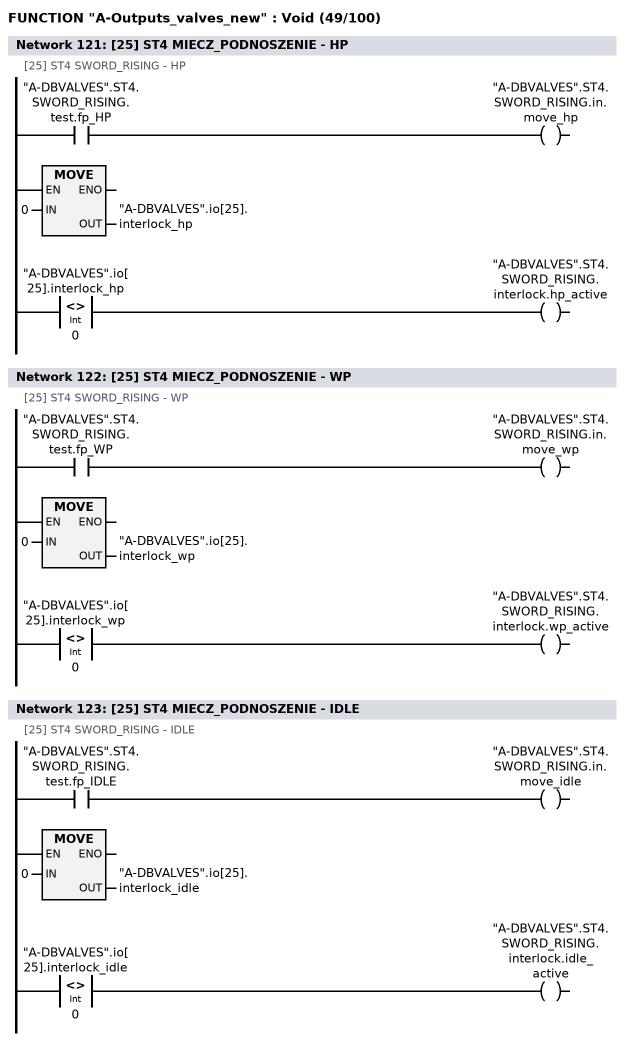
      O "A-DBVALVES".ST4.SWORD_RISING.test.fp_HP;
//    O     "A-Flags".STATION.IN_HP_STEP
      = "A-DBVALVES".ST4.SWORD_RISING.in.move_hp;

// Interlock hp
      L 0;
      T "A-DBVALVES".io[25].interlock_hp;

//{INTERLOCK_HP25}

      A(;
      L "A-DBVALVES".io[25].interlock_hp;
      L 0;
      <>I;
      );
      = "A-DBVALVES".ST4.SWORD_RISING.interlock.hp_active;
NETWORK
TITLE = [25] ST4 MIECZ_PODNOSZENIE - WP
//[25] ST4 SWORD_RISING - WP
      O "A-DBVALVES".ST4.SWORD_RISING.test.fp_WP;
      = "A-DBVALVES".ST4.SWORD_RISING.in.move_wp;

// Interlock wp
      L 0;
      T "A-DBVALVES".io[25].interlock_wp;

//{INTERLOCK_WP25}

      A(;
      L "A-DBVALVES".io[25].interlock_wp;
      L 0;
      <>I;
      );
      = "A-DBVALVES".ST4.SWORD_RISING.interlock.wp_active;
NETWORK
TITLE = [25] ST4 MIECZ_PODNOSZENIE - IDLE
//[25] ST4 SWORD_RISING - IDLE
      O "A-DBVALVES".ST4.SWORD_RISING.test.fp_IDLE;
      = "A-DBVALVES".ST4.SWORD_RISING.in.move_idle;

// Interlock idle
      L 0;
      T "A-DBVALVES".io[25].interlock_idle;

//{INTERLOCK_IDLE25}

      A(;
      L "A-DBVALVES".io[25].interlock_idle;
      L 0;
      <>I;
      );
      = "A-DBVALVES".ST4.SWORD_RISING.interlock.idle_active;
NETWORK
TITLE = [25] ST4 MIECZ_PODNOSZENIE
//[25] ST4 SWORD_RISING
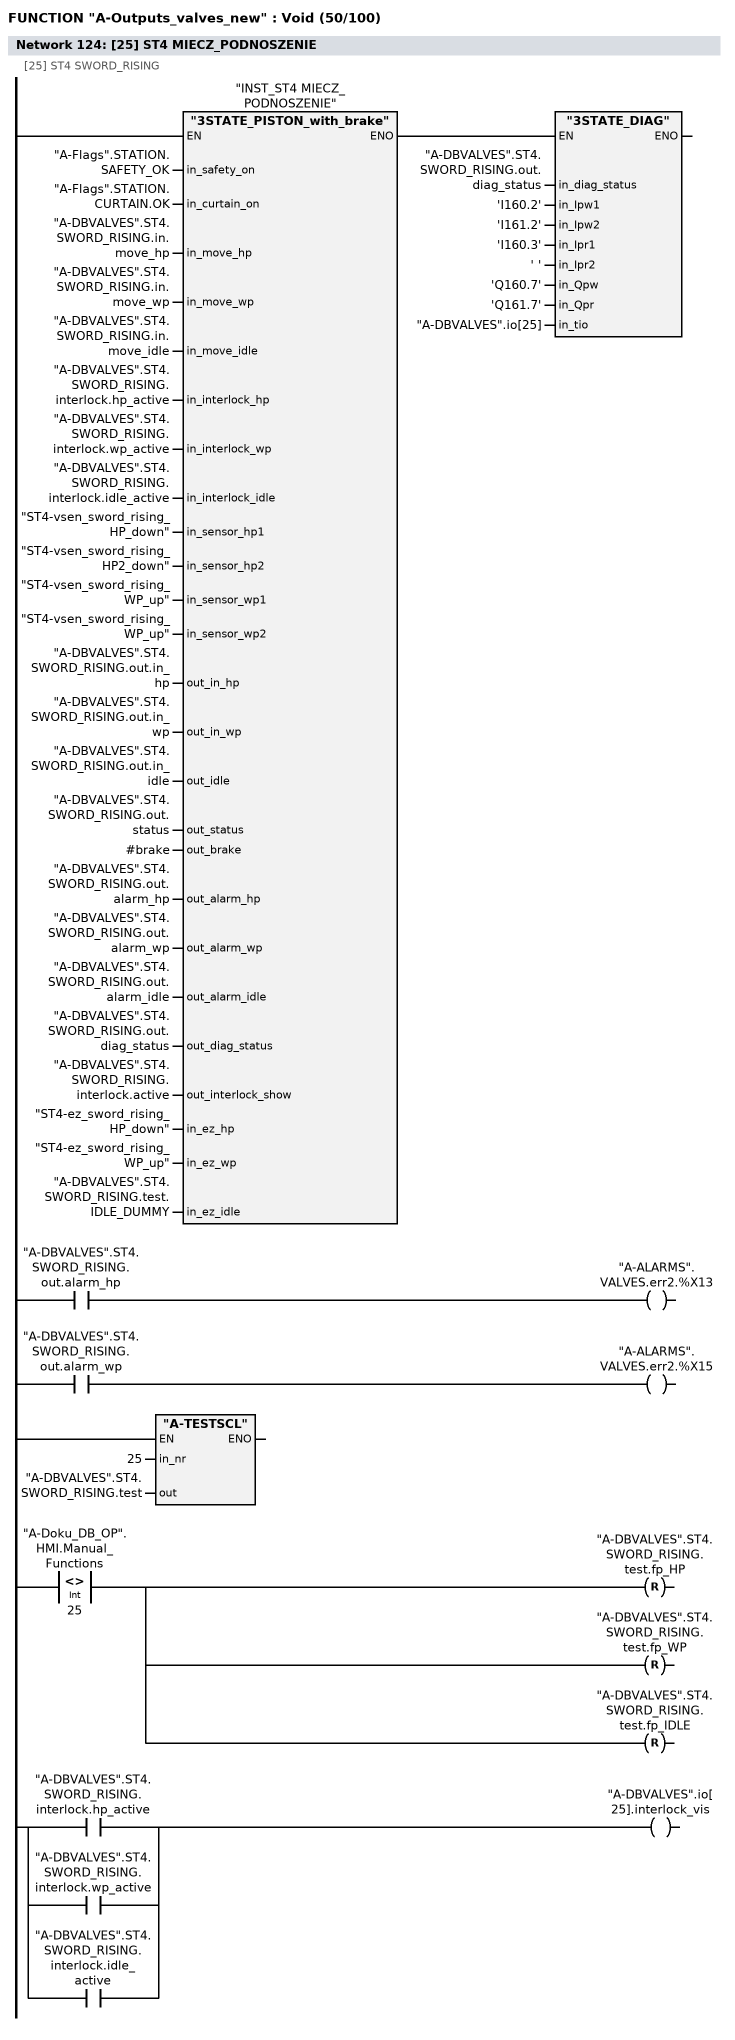
      CALL "3STATE_PISTON_with_brake", "INST_ST4 MIECZ_PODNOSZENIE"
      (  in_safety_on                := "A-Flags".STATION.SAFETY_OK ,
         in_curtain_on               := "A-Flags".STATION.CURTAIN.OK ,
         in_move_hp                  := "A-DBVALVES".ST4.SWORD_RISING.in.move_hp ,
         in_move_wp                  := "A-DBVALVES".ST4.SWORD_RISING.in.move_wp ,
         in_move_idle                := "A-DBVALVES".ST4.SWORD_RISING.in.move_idle ,
         in_interlock_hp             := "A-DBVALVES".ST4.SWORD_RISING.interlock.hp_active ,
         in_interlock_wp             := "A-DBVALVES".ST4.SWORD_RISING.interlock.wp_active ,
         in_interlock_idle           := "A-DBVALVES".ST4.SWORD_RISING.interlock.idle_active ,
         in_sensor_hp1               := "ST4-vsen_sword_rising_HP_down" ,
         in_sensor_hp2               := "ST4-vsen_sword_rising_HP2_down" ,
         in_sensor_wp1               := "ST4-vsen_sword_rising_WP_up" ,
         in_sensor_wp2               := "ST4-vsen_sword_rising_WP_up" ,
         out_in_hp                   := "A-DBVALVES".ST4.SWORD_RISING.out.in_hp ,
         out_in_wp                   := "A-DBVALVES".ST4.SWORD_RISING.out.in_wp ,
         out_idle                    := "A-DBVALVES".ST4.SWORD_RISING.out.in_idle ,
         out_status                  := "A-DBVALVES".ST4.SWORD_RISING.out.status ,
         out_brake                   := #brake ,
         out_alarm_hp                := "A-DBVALVES".ST4.SWORD_RISING.out.alarm_hp ,
         out_alarm_wp                := "A-DBVALVES".ST4.SWORD_RISING.out.alarm_wp ,
         out_alarm_idle              := "A-DBVALVES".ST4.SWORD_RISING.out.alarm_idle ,
         out_diag_status             := "A-DBVALVES".ST4.SWORD_RISING.out.diag_status ,
         out_interlock_show          := "A-DBVALVES".ST4.SWORD_RISING.interlock.active ,
         in_ez_hp                    := "ST4-ez_sword_rising_HP_down" ,
         in_ez_wp                    := "ST4-ez_sword_rising_WP_up" ,
         in_ez_idle                  := "A-DBVALVES".ST4.SWORD_RISING.test.IDLE_DUMMY
      );

      CALL "3STATE_DIAG"
      (  in_diag_status              := "A-DBVALVES".ST4.SWORD_RISING.out.diag_status ,
         in_Ipw1                     := 'I160.2' ,
         in_Ipw2                     := 'I161.2' ,
         in_Ipr1                     := 'I160.3' ,
         in_Ipr2                     := ' ' ,
         in_Qpw                      := 'Q160.7' ,
         in_Qpr                      := 'Q161.7' ,
         in_tio                      := "A-DBVALVES".io[25]
      );

      A "A-DBVALVES".ST4.SWORD_RISING.out.alarm_hp;
      = "A-ALARMS".VALVES.err2.%X13;

      A "A-DBVALVES".ST4.SWORD_RISING.out.alarm_wp;
      = "A-ALARMS".VALVES.err2.%X15;

      CALL "A-TESTSCL"
      (  in_nr                       := 25 ,
         out                         := "A-DBVALVES".ST4.SWORD_RISING.test
      );

      A(;
      L "A-Doku_DB_OP".HMI.Manual_Functions;
      L 25;
      <>I;
      );
      R "A-DBVALVES".ST4.SWORD_RISING.test.fp_HP;
      R "A-DBVALVES".ST4.SWORD_RISING.test.fp_WP;
      R "A-DBVALVES".ST4.SWORD_RISING.test.fp_IDLE;

      O "A-DBVALVES".ST4.SWORD_RISING.interlock.hp_active;
      O "A-DBVALVES".ST4.SWORD_RISING.interlock.wp_active;
      O "A-DBVALVES".ST4.SWORD_RISING.interlock.idle_active;
      = "A-DBVALVES".io[25].interlock_vis;
NETWORK
TITLE = -

NETWORK
TITLE = [26] ST4 ZDERZAK - HP
//[26] ST4 BUMPER - HP
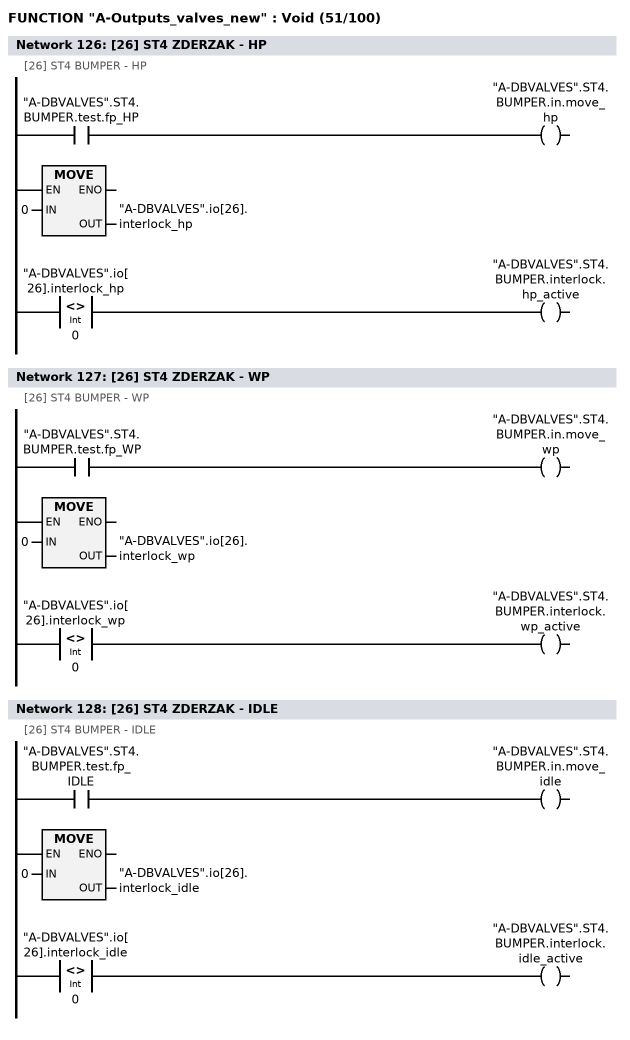
      O "A-DBVALVES".ST4.BUMPER.test.fp_HP;
//    O     "A-Flags".STATION.IN_HP_STEP
      = "A-DBVALVES".ST4.BUMPER.in.move_hp;

// Interlock hp
      L 0;
      T "A-DBVALVES".io[26].interlock_hp;

//{INTERLOCK_HP26}

      A(;
      L "A-DBVALVES".io[26].interlock_hp;
      L 0;
      <>I;
      );
      = "A-DBVALVES".ST4.BUMPER.interlock.hp_active;
NETWORK
TITLE = [26] ST4 ZDERZAK - WP
//[26] ST4 BUMPER - WP
      O "A-DBVALVES".ST4.BUMPER.test.fp_WP;
      = "A-DBVALVES".ST4.BUMPER.in.move_wp;

// Interlock wp
      L 0;
      T "A-DBVALVES".io[26].interlock_wp;

//{INTERLOCK_WP26}

      A(;
      L "A-DBVALVES".io[26].interlock_wp;
      L 0;
      <>I;
      );
      = "A-DBVALVES".ST4.BUMPER.interlock.wp_active;
NETWORK
TITLE = [26] ST4 ZDERZAK - IDLE
//[26] ST4 BUMPER - IDLE
      O "A-DBVALVES".ST4.BUMPER.test.fp_IDLE;
      = "A-DBVALVES".ST4.BUMPER.in.move_idle;

// Interlock idle
      L 0;
      T "A-DBVALVES".io[26].interlock_idle;

//{INTERLOCK_IDLE26}

      A(;
      L "A-DBVALVES".io[26].interlock_idle;
      L 0;
      <>I;
      );
      = "A-DBVALVES".ST4.BUMPER.interlock.idle_active;
NETWORK
TITLE = [26] ST4 ZDERZAK
//[26] ST4 BUMPER
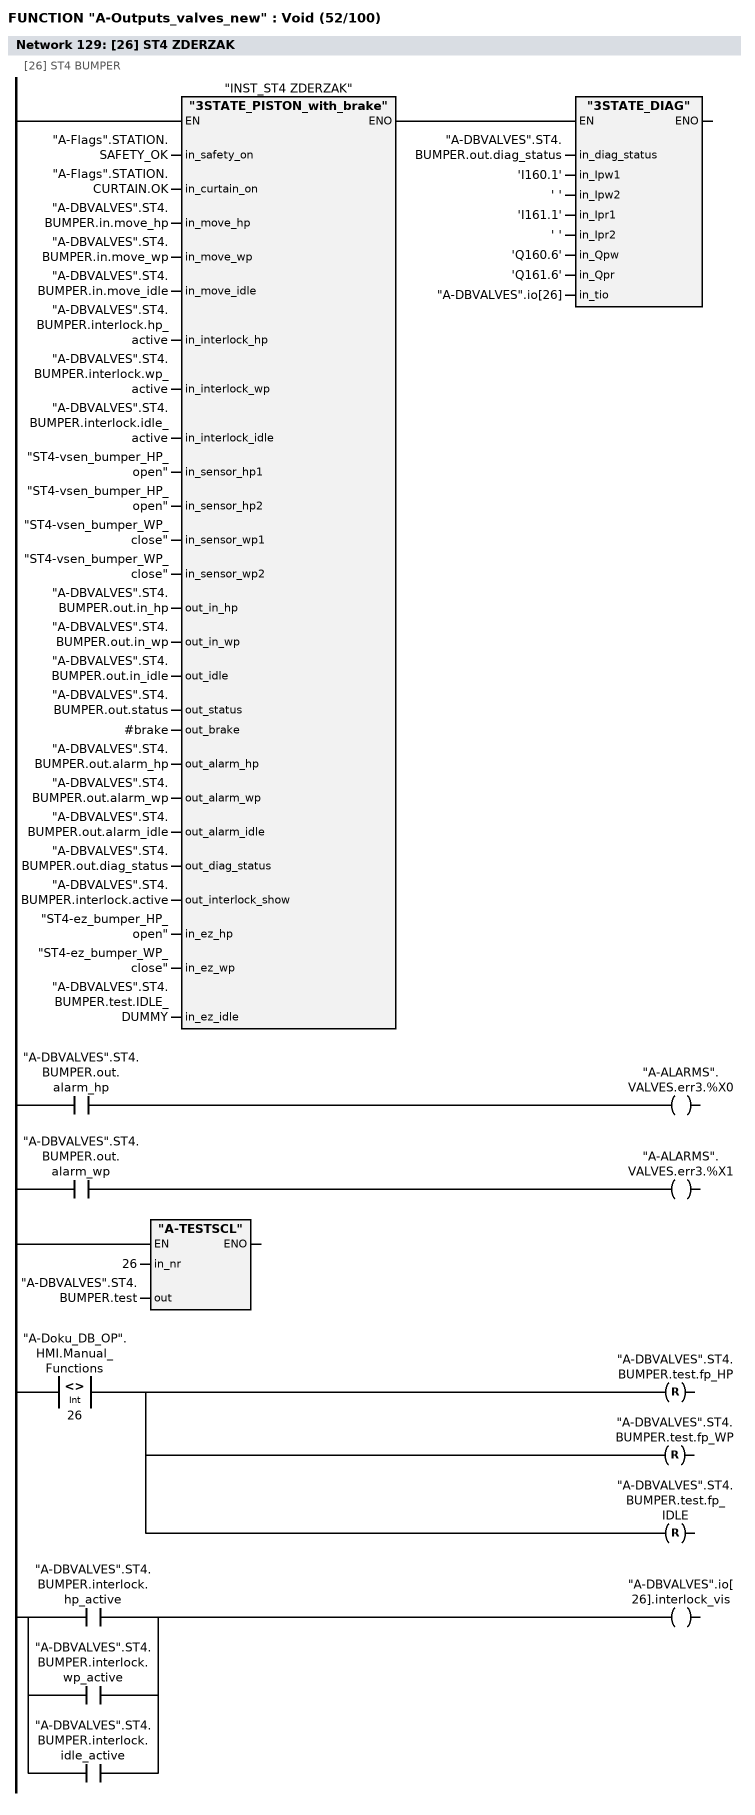
      CALL "3STATE_PISTON_with_brake", "INST_ST4 ZDERZAK"
      (  in_safety_on                := "A-Flags".STATION.SAFETY_OK ,
         in_curtain_on               := "A-Flags".STATION.CURTAIN.OK ,
         in_move_hp                  := "A-DBVALVES".ST4.BUMPER.in.move_hp ,
         in_move_wp                  := "A-DBVALVES".ST4.BUMPER.in.move_wp ,
         in_move_idle                := "A-DBVALVES".ST4.BUMPER.in.move_idle ,
         in_interlock_hp             := "A-DBVALVES".ST4.BUMPER.interlock.hp_active ,
         in_interlock_wp             := "A-DBVALVES".ST4.BUMPER.interlock.wp_active ,
         in_interlock_idle           := "A-DBVALVES".ST4.BUMPER.interlock.idle_active ,
         in_sensor_hp1               := "ST4-vsen_bumper_HP_open" ,
         in_sensor_hp2               := "ST4-vsen_bumper_HP_open" ,
         in_sensor_wp1               := "ST4-vsen_bumper_WP_close" ,
         in_sensor_wp2               := "ST4-vsen_bumper_WP_close" ,
         out_in_hp                   := "A-DBVALVES".ST4.BUMPER.out.in_hp ,
         out_in_wp                   := "A-DBVALVES".ST4.BUMPER.out.in_wp ,
         out_idle                    := "A-DBVALVES".ST4.BUMPER.out.in_idle ,
         out_status                  := "A-DBVALVES".ST4.BUMPER.out.status ,
         out_brake                   := #brake ,
         out_alarm_hp                := "A-DBVALVES".ST4.BUMPER.out.alarm_hp ,
         out_alarm_wp                := "A-DBVALVES".ST4.BUMPER.out.alarm_wp ,
         out_alarm_idle              := "A-DBVALVES".ST4.BUMPER.out.alarm_idle ,
         out_diag_status             := "A-DBVALVES".ST4.BUMPER.out.diag_status ,
         out_interlock_show          := "A-DBVALVES".ST4.BUMPER.interlock.active ,
         in_ez_hp                    := "ST4-ez_bumper_HP_open" ,
         in_ez_wp                    := "ST4-ez_bumper_WP_close" ,
         in_ez_idle                  := "A-DBVALVES".ST4.BUMPER.test.IDLE_DUMMY
      );

      CALL "3STATE_DIAG"
      (  in_diag_status              := "A-DBVALVES".ST4.BUMPER.out.diag_status ,
         in_Ipw1                     := 'I160.1' ,
         in_Ipw2                     := ' ' ,
         in_Ipr1                     := 'I161.1' ,
         in_Ipr2                     := ' ' ,
         in_Qpw                      := 'Q160.6' ,
         in_Qpr                      := 'Q161.6' ,
         in_tio                      := "A-DBVALVES".io[26]
      );

      A "A-DBVALVES".ST4.BUMPER.out.alarm_hp;
      = "A-ALARMS".VALVES.err3.%X0;

      A "A-DBVALVES".ST4.BUMPER.out.alarm_wp;
      = "A-ALARMS".VALVES.err3.%X1;

      CALL "A-TESTSCL"
      (  in_nr                       := 26 ,
         out                         := "A-DBVALVES".ST4.BUMPER.test
      );

      A(;
      L "A-Doku_DB_OP".HMI.Manual_Functions;
      L 26;
      <>I;
      );
      R "A-DBVALVES".ST4.BUMPER.test.fp_HP;
      R "A-DBVALVES".ST4.BUMPER.test.fp_WP;
      R "A-DBVALVES".ST4.BUMPER.test.fp_IDLE;

      O "A-DBVALVES".ST4.BUMPER.interlock.hp_active;
      O "A-DBVALVES".ST4.BUMPER.interlock.wp_active;
      O "A-DBVALVES".ST4.BUMPER.interlock.idle_active;
      = "A-DBVALVES".io[26].interlock_vis;
NETWORK
TITLE = -

NETWORK
TITLE = [27] ST4 MIECZ - HP
//[27] ST4 SWORD - HP
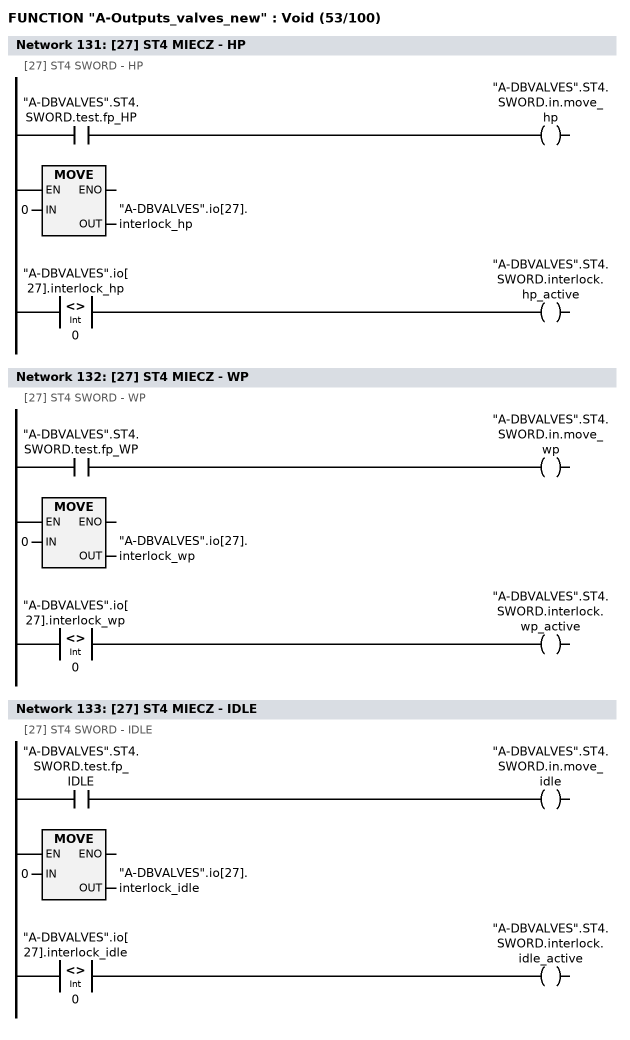
      O "A-DBVALVES".ST4.SWORD.test.fp_HP;
//    O     "A-Flags".STATION.IN_HP_STEP
      = "A-DBVALVES".ST4.SWORD.in.move_hp;

// Interlock hp
      L 0;
      T "A-DBVALVES".io[27].interlock_hp;

//{INTERLOCK_HP27}

      A(;
      L "A-DBVALVES".io[27].interlock_hp;
      L 0;
      <>I;
      );
      = "A-DBVALVES".ST4.SWORD.interlock.hp_active;
NETWORK
TITLE = [27] ST4 MIECZ - WP
//[27] ST4 SWORD - WP
      O "A-DBVALVES".ST4.SWORD.test.fp_WP;
      = "A-DBVALVES".ST4.SWORD.in.move_wp;

// Interlock wp
      L 0;
      T "A-DBVALVES".io[27].interlock_wp;

//{INTERLOCK_WP27}

      A(;
      L "A-DBVALVES".io[27].interlock_wp;
      L 0;
      <>I;
      );
      = "A-DBVALVES".ST4.SWORD.interlock.wp_active;
NETWORK
TITLE = [27] ST4 MIECZ - IDLE
//[27] ST4 SWORD - IDLE
      O "A-DBVALVES".ST4.SWORD.test.fp_IDLE;
      = "A-DBVALVES".ST4.SWORD.in.move_idle;

// Interlock idle
      L 0;
      T "A-DBVALVES".io[27].interlock_idle;

//{INTERLOCK_IDLE27}

      A(;
      L "A-DBVALVES".io[27].interlock_idle;
      L 0;
      <>I;
      );
      = "A-DBVALVES".ST4.SWORD.interlock.idle_active;
NETWORK
TITLE = [27] ST4 MIECZ
//[27] ST4 SWORD
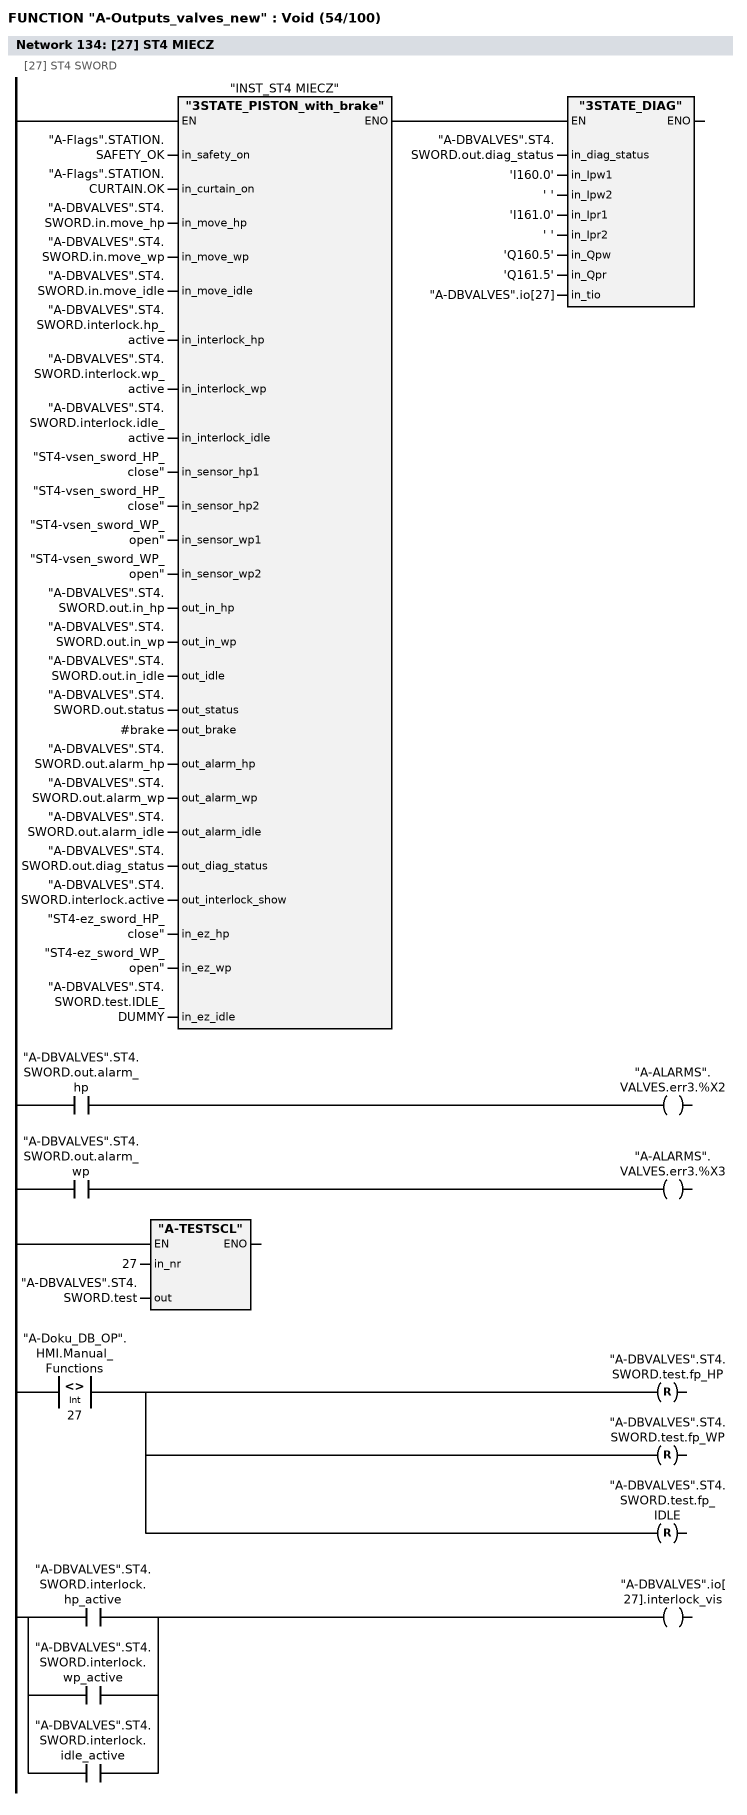
      CALL "3STATE_PISTON_with_brake", "INST_ST4 MIECZ"
      (  in_safety_on                := "A-Flags".STATION.SAFETY_OK ,
         in_curtain_on               := "A-Flags".STATION.CURTAIN.OK ,
         in_move_hp                  := "A-DBVALVES".ST4.SWORD.in.move_hp ,
         in_move_wp                  := "A-DBVALVES".ST4.SWORD.in.move_wp ,
         in_move_idle                := "A-DBVALVES".ST4.SWORD.in.move_idle ,
         in_interlock_hp             := "A-DBVALVES".ST4.SWORD.interlock.hp_active ,
         in_interlock_wp             := "A-DBVALVES".ST4.SWORD.interlock.wp_active ,
         in_interlock_idle           := "A-DBVALVES".ST4.SWORD.interlock.idle_active ,
         in_sensor_hp1               := "ST4-vsen_sword_HP_close" ,
         in_sensor_hp2               := "ST4-vsen_sword_HP_close" ,
         in_sensor_wp1               := "ST4-vsen_sword_WP_open" ,
         in_sensor_wp2               := "ST4-vsen_sword_WP_open" ,
         out_in_hp                   := "A-DBVALVES".ST4.SWORD.out.in_hp ,
         out_in_wp                   := "A-DBVALVES".ST4.SWORD.out.in_wp ,
         out_idle                    := "A-DBVALVES".ST4.SWORD.out.in_idle ,
         out_status                  := "A-DBVALVES".ST4.SWORD.out.status ,
         out_brake                   := #brake ,
         out_alarm_hp                := "A-DBVALVES".ST4.SWORD.out.alarm_hp ,
         out_alarm_wp                := "A-DBVALVES".ST4.SWORD.out.alarm_wp ,
         out_alarm_idle              := "A-DBVALVES".ST4.SWORD.out.alarm_idle ,
         out_diag_status             := "A-DBVALVES".ST4.SWORD.out.diag_status ,
         out_interlock_show          := "A-DBVALVES".ST4.SWORD.interlock.active ,
         in_ez_hp                    := "ST4-ez_sword_HP_close" ,
         in_ez_wp                    := "ST4-ez_sword_WP_open" ,
         in_ez_idle                  := "A-DBVALVES".ST4.SWORD.test.IDLE_DUMMY
      );

      CALL "3STATE_DIAG"
      (  in_diag_status              := "A-DBVALVES".ST4.SWORD.out.diag_status ,
         in_Ipw1                     := 'I160.0' ,
         in_Ipw2                     := ' ' ,
         in_Ipr1                     := 'I161.0' ,
         in_Ipr2                     := ' ' ,
         in_Qpw                      := 'Q160.5' ,
         in_Qpr                      := 'Q161.5' ,
         in_tio                      := "A-DBVALVES".io[27]
      );

      A "A-DBVALVES".ST4.SWORD.out.alarm_hp;
      = "A-ALARMS".VALVES.err3.%X2;

      A "A-DBVALVES".ST4.SWORD.out.alarm_wp;
      = "A-ALARMS".VALVES.err3.%X3;

      CALL "A-TESTSCL"
      (  in_nr                       := 27 ,
         out                         := "A-DBVALVES".ST4.SWORD.test
      );

      A(;
      L "A-Doku_DB_OP".HMI.Manual_Functions;
      L 27;
      <>I;
      );
      R "A-DBVALVES".ST4.SWORD.test.fp_HP;
      R "A-DBVALVES".ST4.SWORD.test.fp_WP;
      R "A-DBVALVES".ST4.SWORD.test.fp_IDLE;

      O "A-DBVALVES".ST4.SWORD.interlock.hp_active;
      O "A-DBVALVES".ST4.SWORD.interlock.wp_active;
      O "A-DBVALVES".ST4.SWORD.interlock.idle_active;
      = "A-DBVALVES".io[27].interlock_vis;
NETWORK
TITLE = -

NETWORK
TITLE = [28] ST5 STACJA_DOJAZD - HP
//[28] ST5 STATION_MOVEMENT - HP
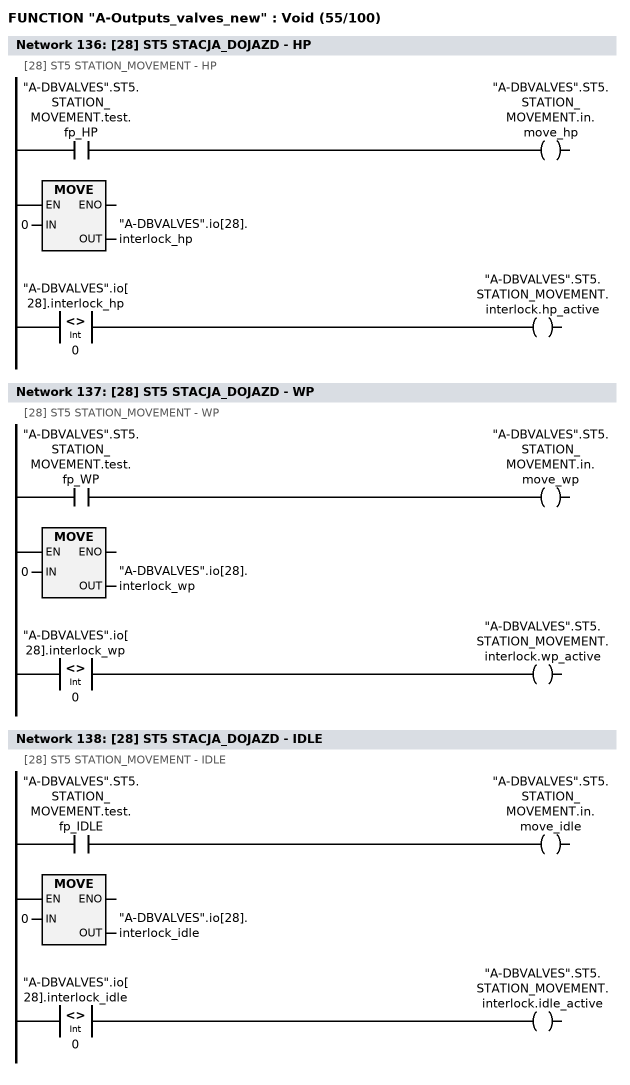
      O "A-DBVALVES".ST5.STATION_MOVEMENT.test.fp_HP;
//    O     "A-Flags".STATION.IN_HP_STEP
      = "A-DBVALVES".ST5.STATION_MOVEMENT.in.move_hp;

// Interlock hp
      L 0;
      T "A-DBVALVES".io[28].interlock_hp;

//{INTERLOCK_HP28}

      A(;
      L "A-DBVALVES".io[28].interlock_hp;
      L 0;
      <>I;
      );
      = "A-DBVALVES".ST5.STATION_MOVEMENT.interlock.hp_active;
NETWORK
TITLE = [28] ST5 STACJA_DOJAZD - WP
//[28] ST5 STATION_MOVEMENT - WP
      O "A-DBVALVES".ST5.STATION_MOVEMENT.test.fp_WP;
      = "A-DBVALVES".ST5.STATION_MOVEMENT.in.move_wp;

// Interlock wp
      L 0;
      T "A-DBVALVES".io[28].interlock_wp;

//{INTERLOCK_WP28}

      A(;
      L "A-DBVALVES".io[28].interlock_wp;
      L 0;
      <>I;
      );
      = "A-DBVALVES".ST5.STATION_MOVEMENT.interlock.wp_active;
NETWORK
TITLE = [28] ST5 STACJA_DOJAZD - IDLE
//[28] ST5 STATION_MOVEMENT - IDLE
      O "A-DBVALVES".ST5.STATION_MOVEMENT.test.fp_IDLE;
      = "A-DBVALVES".ST5.STATION_MOVEMENT.in.move_idle;

// Interlock idle
      L 0;
      T "A-DBVALVES".io[28].interlock_idle;

//{INTERLOCK_IDLE28}

      A(;
      L "A-DBVALVES".io[28].interlock_idle;
      L 0;
      <>I;
      );
      = "A-DBVALVES".ST5.STATION_MOVEMENT.interlock.idle_active;
NETWORK
TITLE = [28] ST5 STACJA_DOJAZD
//[28] ST5 STATION_MOVEMENT
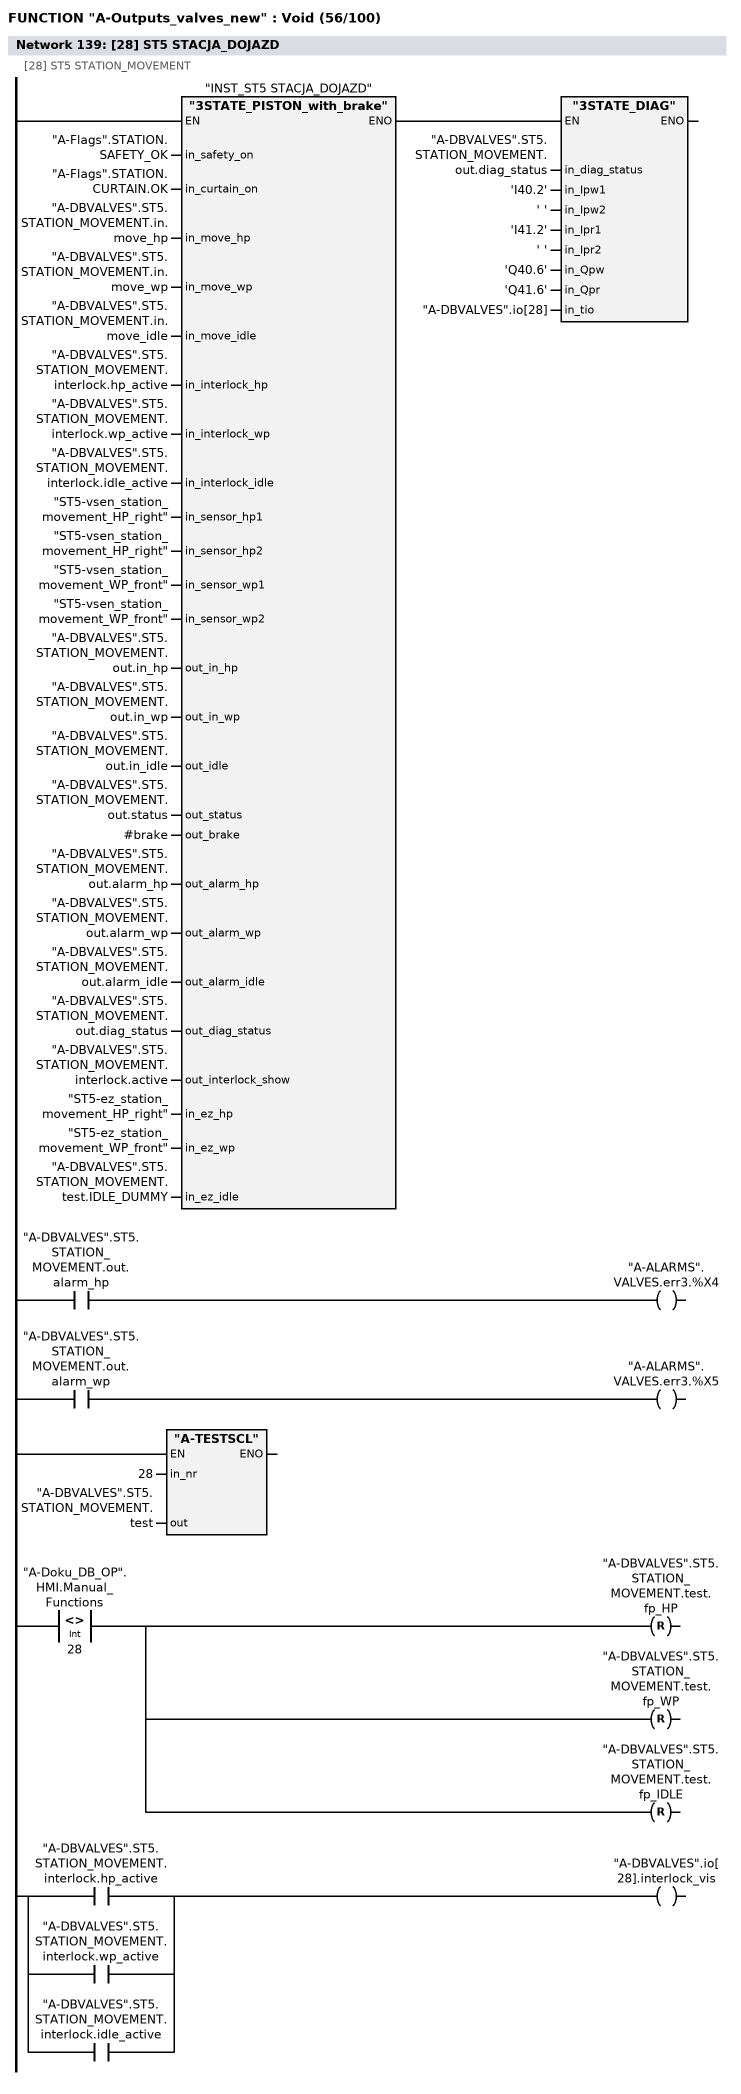
      CALL "3STATE_PISTON_with_brake", "INST_ST5 STACJA_DOJAZD"
      (  in_safety_on                := "A-Flags".STATION.SAFETY_OK ,
         in_curtain_on               := "A-Flags".STATION.CURTAIN.OK ,
         in_move_hp                  := "A-DBVALVES".ST5.STATION_MOVEMENT.in.move_hp ,
         in_move_wp                  := "A-DBVALVES".ST5.STATION_MOVEMENT.in.move_wp ,
         in_move_idle                := "A-DBVALVES".ST5.STATION_MOVEMENT.in.move_idle ,
         in_interlock_hp             := "A-DBVALVES".ST5.STATION_MOVEMENT.interlock.hp_active ,
         in_interlock_wp             := "A-DBVALVES".ST5.STATION_MOVEMENT.interlock.wp_active ,
         in_interlock_idle           := "A-DBVALVES".ST5.STATION_MOVEMENT.interlock.idle_active ,
         in_sensor_hp1               := "ST5-vsen_station_movement_HP_right" ,
         in_sensor_hp2               := "ST5-vsen_station_movement_HP_right" ,
         in_sensor_wp1               := "ST5-vsen_station_movement_WP_front" ,
         in_sensor_wp2               := "ST5-vsen_station_movement_WP_front" ,
         out_in_hp                   := "A-DBVALVES".ST5.STATION_MOVEMENT.out.in_hp ,
         out_in_wp                   := "A-DBVALVES".ST5.STATION_MOVEMENT.out.in_wp ,
         out_idle                    := "A-DBVALVES".ST5.STATION_MOVEMENT.out.in_idle ,
         out_status                  := "A-DBVALVES".ST5.STATION_MOVEMENT.out.status ,
         out_brake                   := #brake ,
         out_alarm_hp                := "A-DBVALVES".ST5.STATION_MOVEMENT.out.alarm_hp ,
         out_alarm_wp                := "A-DBVALVES".ST5.STATION_MOVEMENT.out.alarm_wp ,
         out_alarm_idle              := "A-DBVALVES".ST5.STATION_MOVEMENT.out.alarm_idle ,
         out_diag_status             := "A-DBVALVES".ST5.STATION_MOVEMENT.out.diag_status ,
         out_interlock_show          := "A-DBVALVES".ST5.STATION_MOVEMENT.interlock.active ,
         in_ez_hp                    := "ST5-ez_station_movement_HP_right" ,
         in_ez_wp                    := "ST5-ez_station_movement_WP_front" ,
         in_ez_idle                  := "A-DBVALVES".ST5.STATION_MOVEMENT.test.IDLE_DUMMY
      );

      CALL "3STATE_DIAG"
      (  in_diag_status              := "A-DBVALVES".ST5.STATION_MOVEMENT.out.diag_status ,
         in_Ipw1                     := 'I40.2' ,
         in_Ipw2                     := ' ' ,
         in_Ipr1                     := 'I41.2' ,
         in_Ipr2                     := ' ' ,
         in_Qpw                      := 'Q40.6' ,
         in_Qpr                      := 'Q41.6' ,
         in_tio                      := "A-DBVALVES".io[28]
      );

      A "A-DBVALVES".ST5.STATION_MOVEMENT.out.alarm_hp;
      = "A-ALARMS".VALVES.err3.%X4;

      A "A-DBVALVES".ST5.STATION_MOVEMENT.out.alarm_wp;
      = "A-ALARMS".VALVES.err3.%X5;

      CALL "A-TESTSCL"
      (  in_nr                       := 28 ,
         out                         := "A-DBVALVES".ST5.STATION_MOVEMENT.test
      );

      A(;
      L "A-Doku_DB_OP".HMI.Manual_Functions;
      L 28;
      <>I;
      );
      R "A-DBVALVES".ST5.STATION_MOVEMENT.test.fp_HP;
      R "A-DBVALVES".ST5.STATION_MOVEMENT.test.fp_WP;
      R "A-DBVALVES".ST5.STATION_MOVEMENT.test.fp_IDLE;

      O "A-DBVALVES".ST5.STATION_MOVEMENT.interlock.hp_active;
      O "A-DBVALVES".ST5.STATION_MOVEMENT.interlock.wp_active;
      O "A-DBVALVES".ST5.STATION_MOVEMENT.interlock.idle_active;
      = "A-DBVALVES".io[28].interlock_vis;
NETWORK
TITLE = -

NETWORK
TITLE = [29] ST5 STACJA_MALY_SKOK - HP
//[29] ST5 STATION_SMALL_STEP - HP
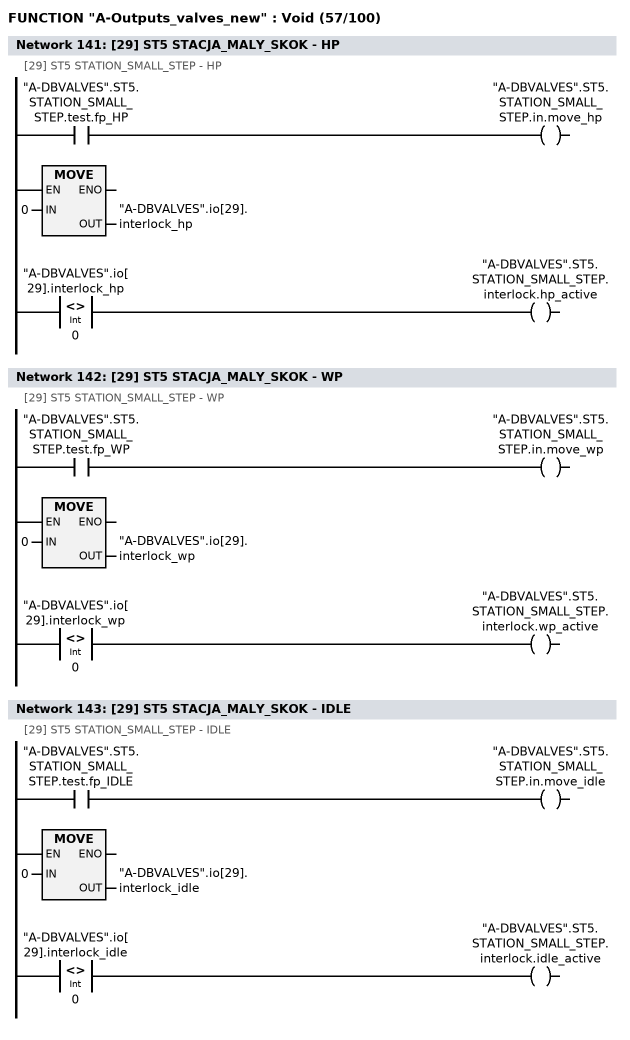
      O "A-DBVALVES".ST5.STATION_SMALL_STEP.test.fp_HP;
//    O     "A-Flags".STATION.IN_HP_STEP
      = "A-DBVALVES".ST5.STATION_SMALL_STEP.in.move_hp;

// Interlock hp
      L 0;
      T "A-DBVALVES".io[29].interlock_hp;

//{INTERLOCK_HP29}

      A(;
      L "A-DBVALVES".io[29].interlock_hp;
      L 0;
      <>I;
      );
      = "A-DBVALVES".ST5.STATION_SMALL_STEP.interlock.hp_active;
NETWORK
TITLE = [29] ST5 STACJA_MALY_SKOK - WP
//[29] ST5 STATION_SMALL_STEP - WP
      O "A-DBVALVES".ST5.STATION_SMALL_STEP.test.fp_WP;
      = "A-DBVALVES".ST5.STATION_SMALL_STEP.in.move_wp;

// Interlock wp
      L 0;
      T "A-DBVALVES".io[29].interlock_wp;

//{INTERLOCK_WP29}

      A(;
      L "A-DBVALVES".io[29].interlock_wp;
      L 0;
      <>I;
      );
      = "A-DBVALVES".ST5.STATION_SMALL_STEP.interlock.wp_active;
NETWORK
TITLE = [29] ST5 STACJA_MALY_SKOK - IDLE
//[29] ST5 STATION_SMALL_STEP - IDLE
      O "A-DBVALVES".ST5.STATION_SMALL_STEP.test.fp_IDLE;
      = "A-DBVALVES".ST5.STATION_SMALL_STEP.in.move_idle;

// Interlock idle
      L 0;
      T "A-DBVALVES".io[29].interlock_idle;

//{INTERLOCK_IDLE29}

      A(;
      L "A-DBVALVES".io[29].interlock_idle;
      L 0;
      <>I;
      );
      = "A-DBVALVES".ST5.STATION_SMALL_STEP.interlock.idle_active;
NETWORK
TITLE = [29] ST5 STACJA_MALY_SKOK
//[29] ST5 STATION_SMALL_STEP
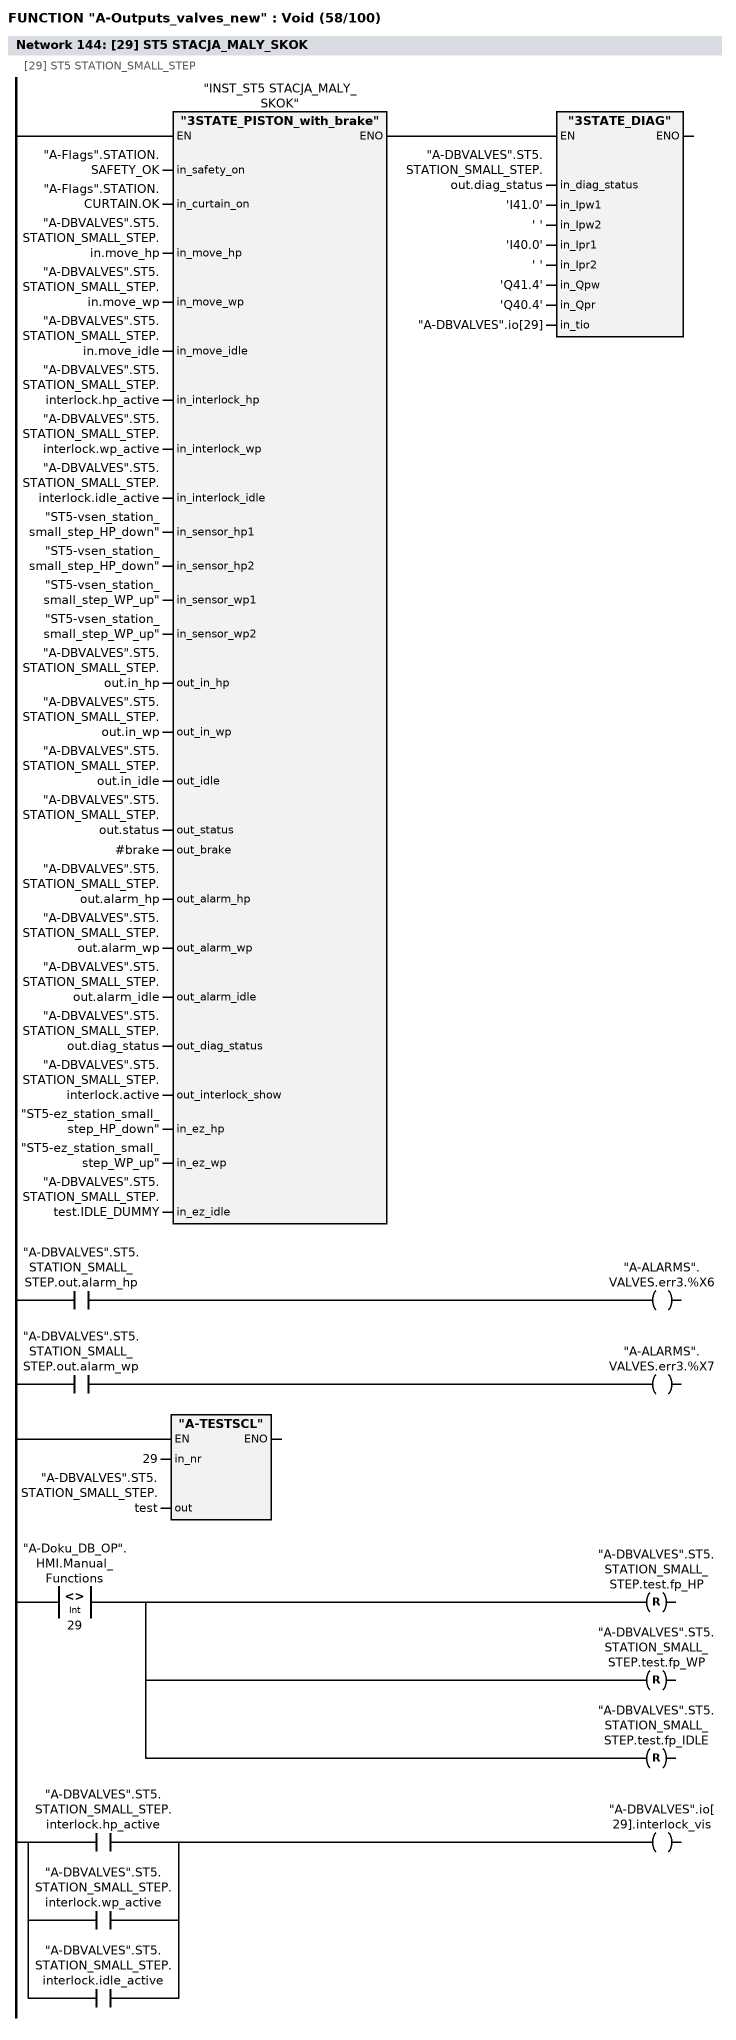
      CALL "3STATE_PISTON_with_brake", "INST_ST5 STACJA_MALY_SKOK"
      (  in_safety_on                := "A-Flags".STATION.SAFETY_OK ,
         in_curtain_on               := "A-Flags".STATION.CURTAIN.OK ,
         in_move_hp                  := "A-DBVALVES".ST5.STATION_SMALL_STEP.in.move_hp ,
         in_move_wp                  := "A-DBVALVES".ST5.STATION_SMALL_STEP.in.move_wp ,
         in_move_idle                := "A-DBVALVES".ST5.STATION_SMALL_STEP.in.move_idle ,
         in_interlock_hp             := "A-DBVALVES".ST5.STATION_SMALL_STEP.interlock.hp_active ,
         in_interlock_wp             := "A-DBVALVES".ST5.STATION_SMALL_STEP.interlock.wp_active ,
         in_interlock_idle           := "A-DBVALVES".ST5.STATION_SMALL_STEP.interlock.idle_active ,
         in_sensor_hp1               := "ST5-vsen_station_small_step_HP_down" ,
         in_sensor_hp2               := "ST5-vsen_station_small_step_HP_down" ,
         in_sensor_wp1               := "ST5-vsen_station_small_step_WP_up" ,
         in_sensor_wp2               := "ST5-vsen_station_small_step_WP_up" ,
         out_in_hp                   := "A-DBVALVES".ST5.STATION_SMALL_STEP.out.in_hp ,
         out_in_wp                   := "A-DBVALVES".ST5.STATION_SMALL_STEP.out.in_wp ,
         out_idle                    := "A-DBVALVES".ST5.STATION_SMALL_STEP.out.in_idle ,
         out_status                  := "A-DBVALVES".ST5.STATION_SMALL_STEP.out.status ,
         out_brake                   := #brake ,
         out_alarm_hp                := "A-DBVALVES".ST5.STATION_SMALL_STEP.out.alarm_hp ,
         out_alarm_wp                := "A-DBVALVES".ST5.STATION_SMALL_STEP.out.alarm_wp ,
         out_alarm_idle              := "A-DBVALVES".ST5.STATION_SMALL_STEP.out.alarm_idle ,
         out_diag_status             := "A-DBVALVES".ST5.STATION_SMALL_STEP.out.diag_status ,
         out_interlock_show          := "A-DBVALVES".ST5.STATION_SMALL_STEP.interlock.active ,
         in_ez_hp                    := "ST5-ez_station_small_step_HP_down" ,
         in_ez_wp                    := "ST5-ez_station_small_step_WP_up" ,
         in_ez_idle                  := "A-DBVALVES".ST5.STATION_SMALL_STEP.test.IDLE_DUMMY
      );

      CALL "3STATE_DIAG"
      (  in_diag_status              := "A-DBVALVES".ST5.STATION_SMALL_STEP.out.diag_status ,
         in_Ipw1                     := 'I41.0' ,
         in_Ipw2                     := ' ' ,
         in_Ipr1                     := 'I40.0' ,
         in_Ipr2                     := ' ' ,
         in_Qpw                      := 'Q41.4' ,
         in_Qpr                      := 'Q40.4' ,
         in_tio                      := "A-DBVALVES".io[29]
      );

      A "A-DBVALVES".ST5.STATION_SMALL_STEP.out.alarm_hp;
      = "A-ALARMS".VALVES.err3.%X6;

      A "A-DBVALVES".ST5.STATION_SMALL_STEP.out.alarm_wp;
      = "A-ALARMS".VALVES.err3.%X7;

      CALL "A-TESTSCL"
      (  in_nr                       := 29 ,
         out                         := "A-DBVALVES".ST5.STATION_SMALL_STEP.test
      );

      A(;
      L "A-Doku_DB_OP".HMI.Manual_Functions;
      L 29;
      <>I;
      );
      R "A-DBVALVES".ST5.STATION_SMALL_STEP.test.fp_HP;
      R "A-DBVALVES".ST5.STATION_SMALL_STEP.test.fp_WP;
      R "A-DBVALVES".ST5.STATION_SMALL_STEP.test.fp_IDLE;

      O "A-DBVALVES".ST5.STATION_SMALL_STEP.interlock.hp_active;
      O "A-DBVALVES".ST5.STATION_SMALL_STEP.interlock.wp_active;
      O "A-DBVALVES".ST5.STATION_SMALL_STEP.interlock.idle_active;
      = "A-DBVALVES".io[29].interlock_vis;
NETWORK
TITLE = -

NETWORK
TITLE = [30] ST5 STACJA_DUZY_SKOK - HP
//[30] ST5 STATION_BIG_STEP - HP
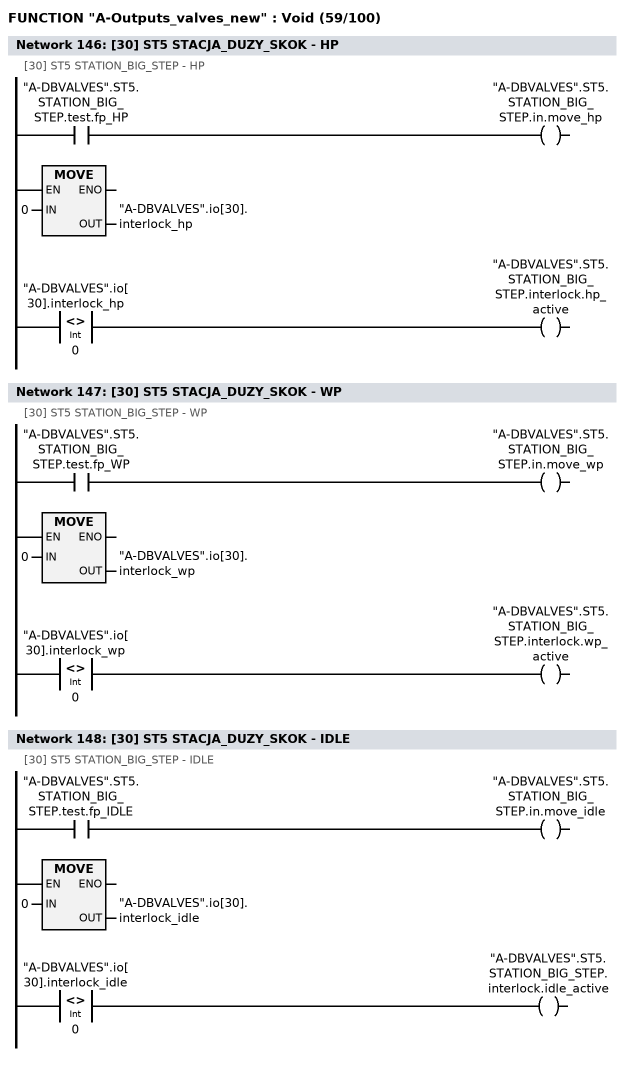
      O "A-DBVALVES".ST5.STATION_BIG_STEP.test.fp_HP;
//    O     "A-Flags".STATION.IN_HP_STEP
      = "A-DBVALVES".ST5.STATION_BIG_STEP.in.move_hp;

// Interlock hp
      L 0;
      T "A-DBVALVES".io[30].interlock_hp;

//{INTERLOCK_HP30}

      A(;
      L "A-DBVALVES".io[30].interlock_hp;
      L 0;
      <>I;
      );
      = "A-DBVALVES".ST5.STATION_BIG_STEP.interlock.hp_active;
NETWORK
TITLE = [30] ST5 STACJA_DUZY_SKOK - WP
//[30] ST5 STATION_BIG_STEP - WP
      O "A-DBVALVES".ST5.STATION_BIG_STEP.test.fp_WP;
      = "A-DBVALVES".ST5.STATION_BIG_STEP.in.move_wp;

// Interlock wp
      L 0;
      T "A-DBVALVES".io[30].interlock_wp;

//{INTERLOCK_WP30}

      A(;
      L "A-DBVALVES".io[30].interlock_wp;
      L 0;
      <>I;
      );
      = "A-DBVALVES".ST5.STATION_BIG_STEP.interlock.wp_active;
NETWORK
TITLE = [30] ST5 STACJA_DUZY_SKOK - IDLE
//[30] ST5 STATION_BIG_STEP - IDLE
      O "A-DBVALVES".ST5.STATION_BIG_STEP.test.fp_IDLE;
      = "A-DBVALVES".ST5.STATION_BIG_STEP.in.move_idle;

// Interlock idle
      L 0;
      T "A-DBVALVES".io[30].interlock_idle;

//{INTERLOCK_IDLE30}

      A(;
      L "A-DBVALVES".io[30].interlock_idle;
      L 0;
      <>I;
      );
      = "A-DBVALVES".ST5.STATION_BIG_STEP.interlock.idle_active;
NETWORK
TITLE = [30] ST5 STACJA_DUZY_SKOK
//[30] ST5 STATION_BIG_STEP
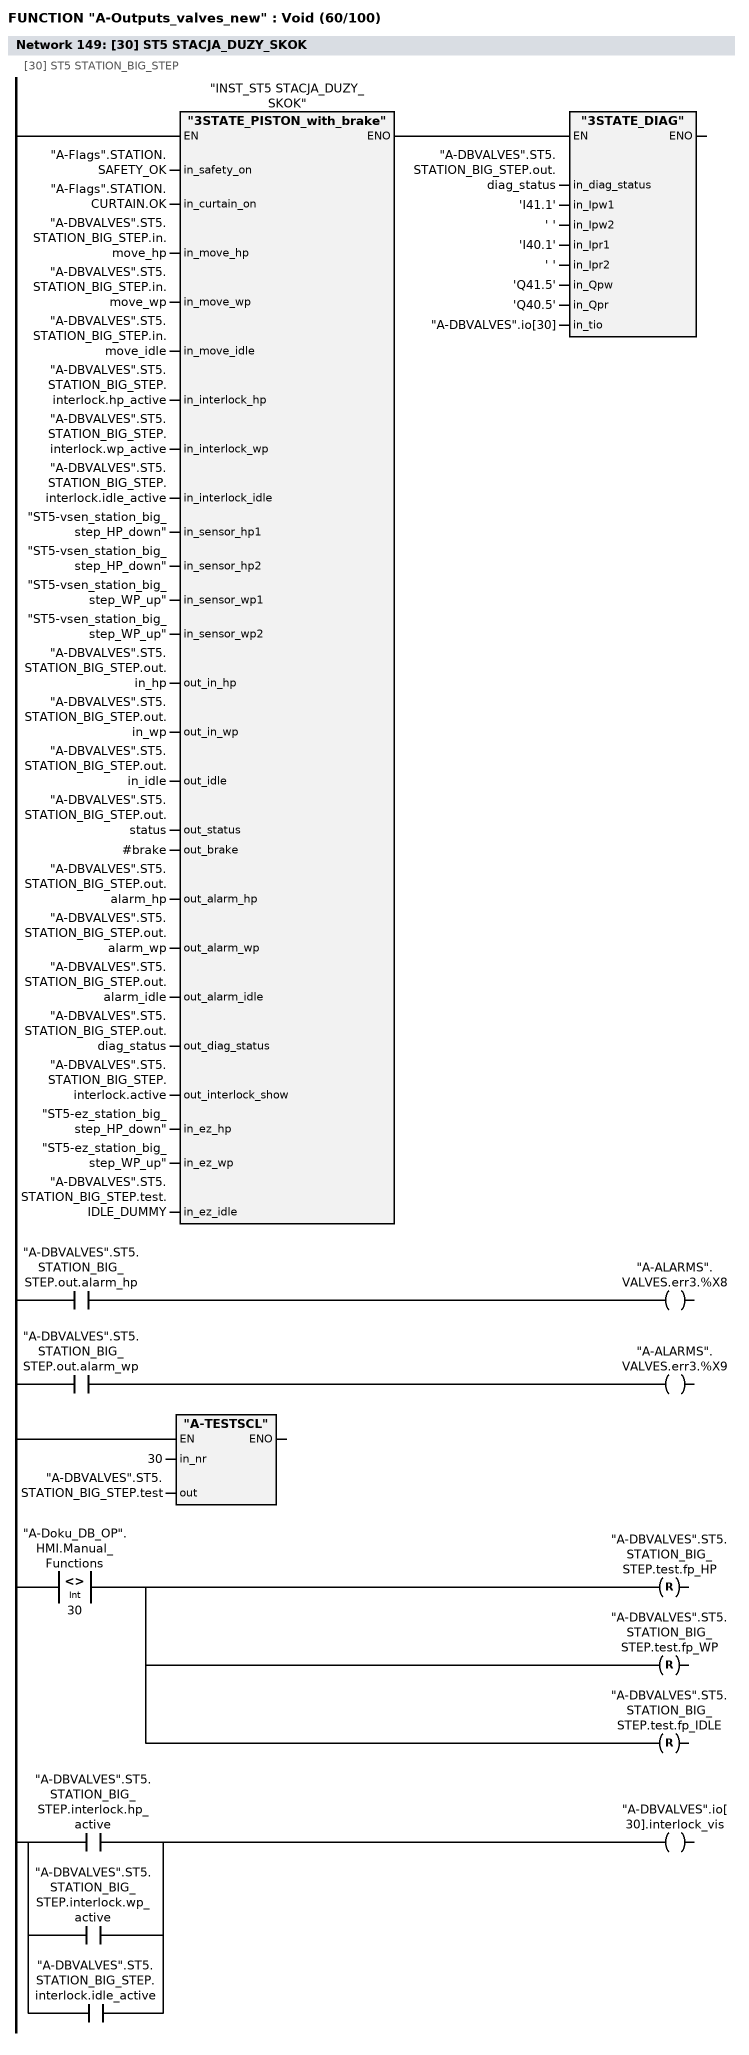
      CALL "3STATE_PISTON_with_brake", "INST_ST5 STACJA_DUZY_SKOK"
      (  in_safety_on                := "A-Flags".STATION.SAFETY_OK ,
         in_curtain_on               := "A-Flags".STATION.CURTAIN.OK ,
         in_move_hp                  := "A-DBVALVES".ST5.STATION_BIG_STEP.in.move_hp ,
         in_move_wp                  := "A-DBVALVES".ST5.STATION_BIG_STEP.in.move_wp ,
         in_move_idle                := "A-DBVALVES".ST5.STATION_BIG_STEP.in.move_idle ,
         in_interlock_hp             := "A-DBVALVES".ST5.STATION_BIG_STEP.interlock.hp_active ,
         in_interlock_wp             := "A-DBVALVES".ST5.STATION_BIG_STEP.interlock.wp_active ,
         in_interlock_idle           := "A-DBVALVES".ST5.STATION_BIG_STEP.interlock.idle_active ,
         in_sensor_hp1               := "ST5-vsen_station_big_step_HP_down" ,
         in_sensor_hp2               := "ST5-vsen_station_big_step_HP_down" ,
         in_sensor_wp1               := "ST5-vsen_station_big_step_WP_up" ,
         in_sensor_wp2               := "ST5-vsen_station_big_step_WP_up" ,
         out_in_hp                   := "A-DBVALVES".ST5.STATION_BIG_STEP.out.in_hp ,
         out_in_wp                   := "A-DBVALVES".ST5.STATION_BIG_STEP.out.in_wp ,
         out_idle                    := "A-DBVALVES".ST5.STATION_BIG_STEP.out.in_idle ,
         out_status                  := "A-DBVALVES".ST5.STATION_BIG_STEP.out.status ,
         out_brake                   := #brake ,
         out_alarm_hp                := "A-DBVALVES".ST5.STATION_BIG_STEP.out.alarm_hp ,
         out_alarm_wp                := "A-DBVALVES".ST5.STATION_BIG_STEP.out.alarm_wp ,
         out_alarm_idle              := "A-DBVALVES".ST5.STATION_BIG_STEP.out.alarm_idle ,
         out_diag_status             := "A-DBVALVES".ST5.STATION_BIG_STEP.out.diag_status ,
         out_interlock_show          := "A-DBVALVES".ST5.STATION_BIG_STEP.interlock.active ,
         in_ez_hp                    := "ST5-ez_station_big_step_HP_down" ,
         in_ez_wp                    := "ST5-ez_station_big_step_WP_up" ,
         in_ez_idle                  := "A-DBVALVES".ST5.STATION_BIG_STEP.test.IDLE_DUMMY
      );

      CALL "3STATE_DIAG"
      (  in_diag_status              := "A-DBVALVES".ST5.STATION_BIG_STEP.out.diag_status ,
         in_Ipw1                     := 'I41.1' ,
         in_Ipw2                     := ' ' ,
         in_Ipr1                     := 'I40.1' ,
         in_Ipr2                     := ' ' ,
         in_Qpw                      := 'Q41.5' ,
         in_Qpr                      := 'Q40.5' ,
         in_tio                      := "A-DBVALVES".io[30]
      );

      A "A-DBVALVES".ST5.STATION_BIG_STEP.out.alarm_hp;
      = "A-ALARMS".VALVES.err3.%X8;

      A "A-DBVALVES".ST5.STATION_BIG_STEP.out.alarm_wp;
      = "A-ALARMS".VALVES.err3.%X9;

      CALL "A-TESTSCL"
      (  in_nr                       := 30 ,
         out                         := "A-DBVALVES".ST5.STATION_BIG_STEP.test
      );

      A(;
      L "A-Doku_DB_OP".HMI.Manual_Functions;
      L 30;
      <>I;
      );
      R "A-DBVALVES".ST5.STATION_BIG_STEP.test.fp_HP;
      R "A-DBVALVES".ST5.STATION_BIG_STEP.test.fp_WP;
      R "A-DBVALVES".ST5.STATION_BIG_STEP.test.fp_IDLE;

      O "A-DBVALVES".ST5.STATION_BIG_STEP.interlock.hp_active;
      O "A-DBVALVES".ST5.STATION_BIG_STEP.interlock.wp_active;
      O "A-DBVALVES".ST5.STATION_BIG_STEP.interlock.idle_active;
      = "A-DBVALVES".io[30].interlock_vis;
NETWORK
TITLE = -

NETWORK
TITLE = [31] ST5 PIN - HP
//[31] ST5 PIN - HP
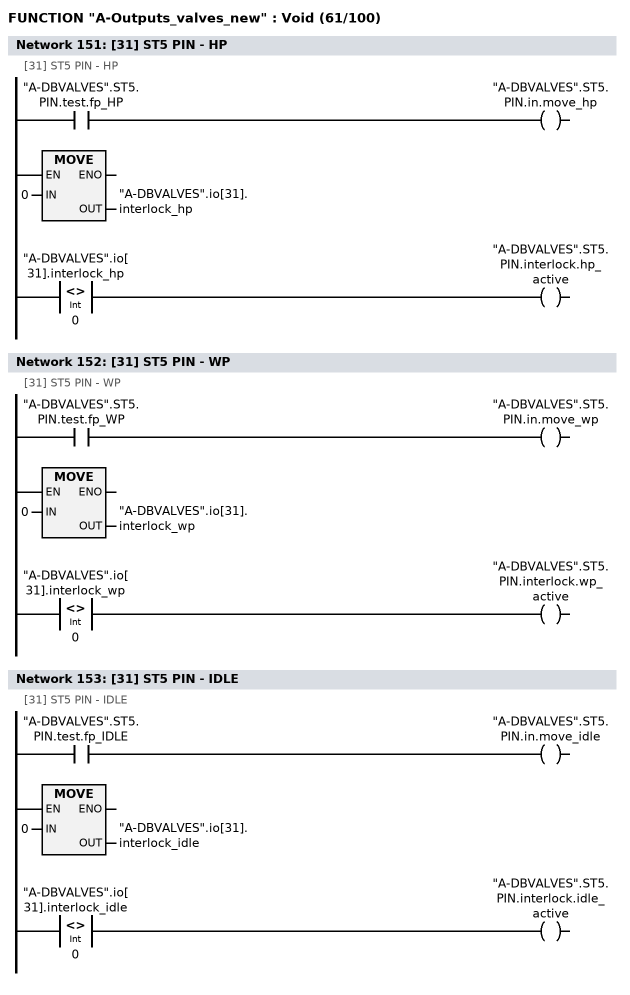
      O "A-DBVALVES".ST5.PIN.test.fp_HP;
//    O     "A-Flags".STATION.IN_HP_STEP
      = "A-DBVALVES".ST5.PIN.in.move_hp;

// Interlock hp
      L 0;
      T "A-DBVALVES".io[31].interlock_hp;

//{INTERLOCK_HP31}

      A(;
      L "A-DBVALVES".io[31].interlock_hp;
      L 0;
      <>I;
      );
      = "A-DBVALVES".ST5.PIN.interlock.hp_active;
NETWORK
TITLE = [31] ST5 PIN - WP
//[31] ST5 PIN - WP
      O "A-DBVALVES".ST5.PIN.test.fp_WP;
      = "A-DBVALVES".ST5.PIN.in.move_wp;

// Interlock wp
      L 0;
      T "A-DBVALVES".io[31].interlock_wp;

//{INTERLOCK_WP31}

      A(;
      L "A-DBVALVES".io[31].interlock_wp;
      L 0;
      <>I;
      );
      = "A-DBVALVES".ST5.PIN.interlock.wp_active;
NETWORK
TITLE = [31] ST5 PIN - IDLE
//[31] ST5 PIN - IDLE
      O "A-DBVALVES".ST5.PIN.test.fp_IDLE;
      = "A-DBVALVES".ST5.PIN.in.move_idle;

// Interlock idle
      L 0;
      T "A-DBVALVES".io[31].interlock_idle;

//{INTERLOCK_IDLE31}

      A(;
      L "A-DBVALVES".io[31].interlock_idle;
      L 0;
      <>I;
      );
      = "A-DBVALVES".ST5.PIN.interlock.idle_active;
NETWORK
TITLE = [31] ST5 PIN
//[31] ST5 PIN
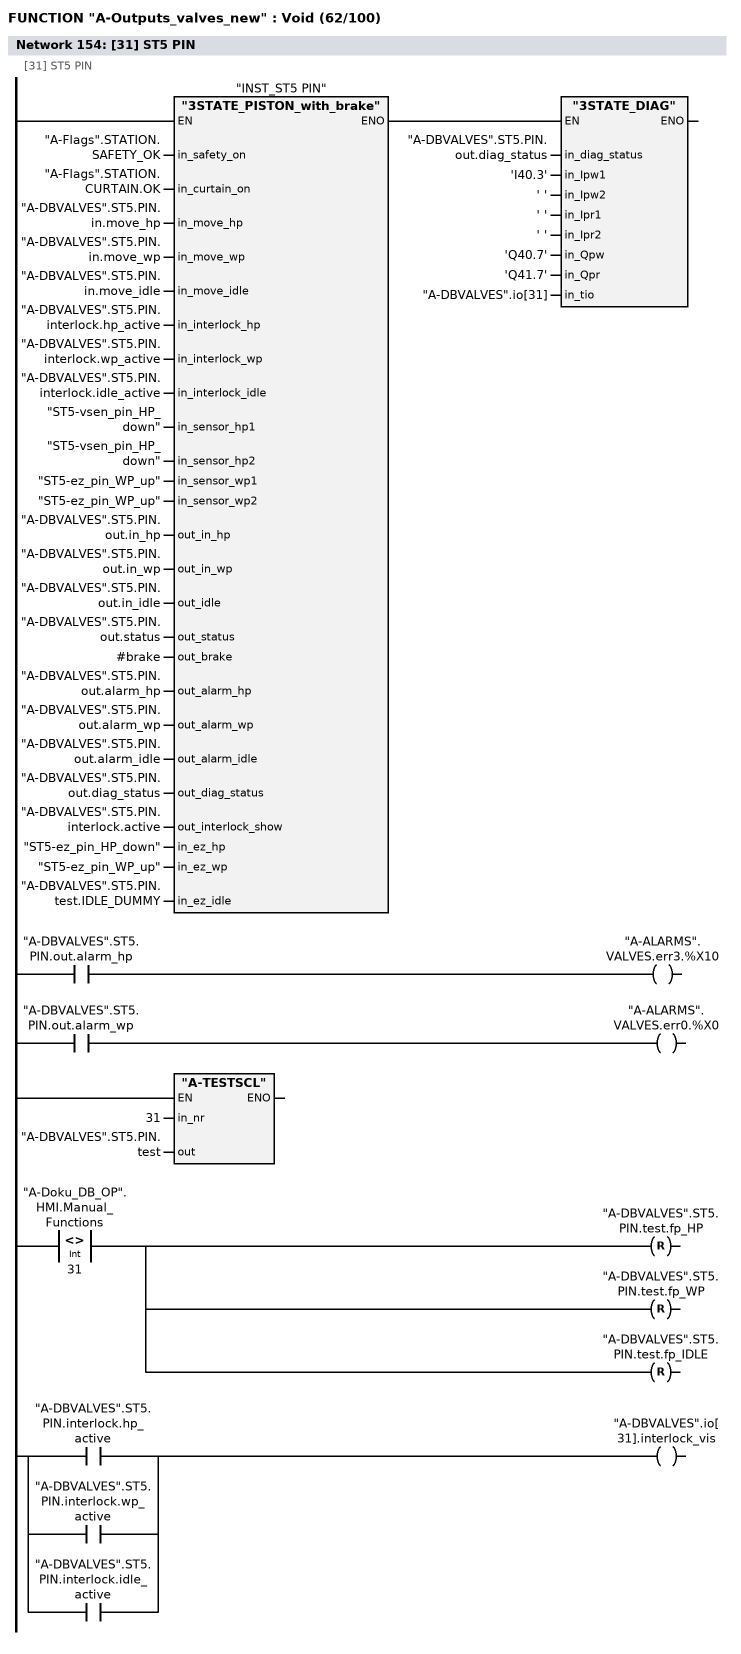
      CALL "3STATE_PISTON_with_brake", "INST_ST5 PIN"
      (  in_safety_on                := "A-Flags".STATION.SAFETY_OK ,
         in_curtain_on               := "A-Flags".STATION.CURTAIN.OK ,
         in_move_hp                  := "A-DBVALVES".ST5.PIN.in.move_hp ,
         in_move_wp                  := "A-DBVALVES".ST5.PIN.in.move_wp ,
         in_move_idle                := "A-DBVALVES".ST5.PIN.in.move_idle ,
         in_interlock_hp             := "A-DBVALVES".ST5.PIN.interlock.hp_active ,
         in_interlock_wp             := "A-DBVALVES".ST5.PIN.interlock.wp_active ,
         in_interlock_idle           := "A-DBVALVES".ST5.PIN.interlock.idle_active ,
         in_sensor_hp1               := "ST5-vsen_pin_HP_down" ,
         in_sensor_hp2               := "ST5-vsen_pin_HP_down" ,
         in_sensor_wp1               := "ST5-ez_pin_WP_up" ,
         in_sensor_wp2               := "ST5-ez_pin_WP_up" ,
         out_in_hp                   := "A-DBVALVES".ST5.PIN.out.in_hp ,
         out_in_wp                   := "A-DBVALVES".ST5.PIN.out.in_wp ,
         out_idle                    := "A-DBVALVES".ST5.PIN.out.in_idle ,
         out_status                  := "A-DBVALVES".ST5.PIN.out.status ,
         out_brake                   := #brake ,
         out_alarm_hp                := "A-DBVALVES".ST5.PIN.out.alarm_hp ,
         out_alarm_wp                := "A-DBVALVES".ST5.PIN.out.alarm_wp ,
         out_alarm_idle              := "A-DBVALVES".ST5.PIN.out.alarm_idle ,
         out_diag_status             := "A-DBVALVES".ST5.PIN.out.diag_status ,
         out_interlock_show          := "A-DBVALVES".ST5.PIN.interlock.active ,
         in_ez_hp                    := "ST5-ez_pin_HP_down" ,
         in_ez_wp                    := "ST5-ez_pin_WP_up" ,
         in_ez_idle                  := "A-DBVALVES".ST5.PIN.test.IDLE_DUMMY
      );

      CALL "3STATE_DIAG"
      (  in_diag_status              := "A-DBVALVES".ST5.PIN.out.diag_status ,
         in_Ipw1                     := 'I40.3' ,
         in_Ipw2                     := ' ' ,
         in_Ipr1                     := ' ' ,
         in_Ipr2                     := ' ' ,
         in_Qpw                      := 'Q40.7' ,
         in_Qpr                      := 'Q41.7' ,
         in_tio                      := "A-DBVALVES".io[31]
      );

      A "A-DBVALVES".ST5.PIN.out.alarm_hp;
      = "A-ALARMS".VALVES.err3.%X10;

      A "A-DBVALVES".ST5.PIN.out.alarm_wp;
      = "A-ALARMS".VALVES.err0.%X0;

      CALL "A-TESTSCL"
      (  in_nr                       := 31 ,
         out                         := "A-DBVALVES".ST5.PIN.test
      );

      A(;
      L "A-Doku_DB_OP".HMI.Manual_Functions;
      L 31;
      <>I;
      );
      R "A-DBVALVES".ST5.PIN.test.fp_HP;
      R "A-DBVALVES".ST5.PIN.test.fp_WP;
      R "A-DBVALVES".ST5.PIN.test.fp_IDLE;

      O "A-DBVALVES".ST5.PIN.interlock.hp_active;
      O "A-DBVALVES".ST5.PIN.interlock.wp_active;
      O "A-DBVALVES".ST5.PIN.interlock.idle_active;
      = "A-DBVALVES".io[31].interlock_vis;
NETWORK
TITLE = -

NETWORK
TITLE = [32] ST6 STACJA_DOJAZD - HP
//[32] ST6 STATION_MOVEMENT - HP
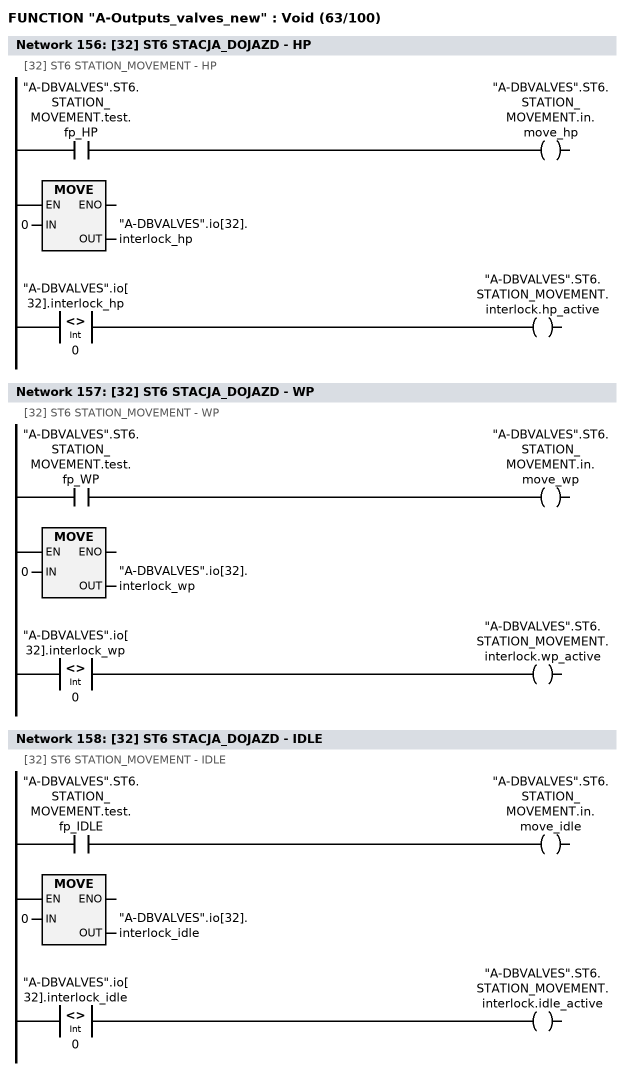
      O "A-DBVALVES".ST6.STATION_MOVEMENT.test.fp_HP;
//    O     "A-Flags".STATION.IN_HP_STEP
      = "A-DBVALVES".ST6.STATION_MOVEMENT.in.move_hp;

// Interlock hp
      L 0;
      T "A-DBVALVES".io[32].interlock_hp;

//{INTERLOCK_HP32}

      A(;
      L "A-DBVALVES".io[32].interlock_hp;
      L 0;
      <>I;
      );
      = "A-DBVALVES".ST6.STATION_MOVEMENT.interlock.hp_active;
NETWORK
TITLE = [32] ST6 STACJA_DOJAZD - WP
//[32] ST6 STATION_MOVEMENT - WP
      O "A-DBVALVES".ST6.STATION_MOVEMENT.test.fp_WP;
      = "A-DBVALVES".ST6.STATION_MOVEMENT.in.move_wp;

// Interlock wp
      L 0;
      T "A-DBVALVES".io[32].interlock_wp;

//{INTERLOCK_WP32}

      A(;
      L "A-DBVALVES".io[32].interlock_wp;
      L 0;
      <>I;
      );
      = "A-DBVALVES".ST6.STATION_MOVEMENT.interlock.wp_active;
NETWORK
TITLE = [32] ST6 STACJA_DOJAZD - IDLE
//[32] ST6 STATION_MOVEMENT - IDLE
      O "A-DBVALVES".ST6.STATION_MOVEMENT.test.fp_IDLE;
      = "A-DBVALVES".ST6.STATION_MOVEMENT.in.move_idle;

// Interlock idle
      L 0;
      T "A-DBVALVES".io[32].interlock_idle;

//{INTERLOCK_IDLE32}

      A(;
      L "A-DBVALVES".io[32].interlock_idle;
      L 0;
      <>I;
      );
      = "A-DBVALVES".ST6.STATION_MOVEMENT.interlock.idle_active;
NETWORK
TITLE = [32] ST6 STACJA_DOJAZD
//[32] ST6 STATION_MOVEMENT
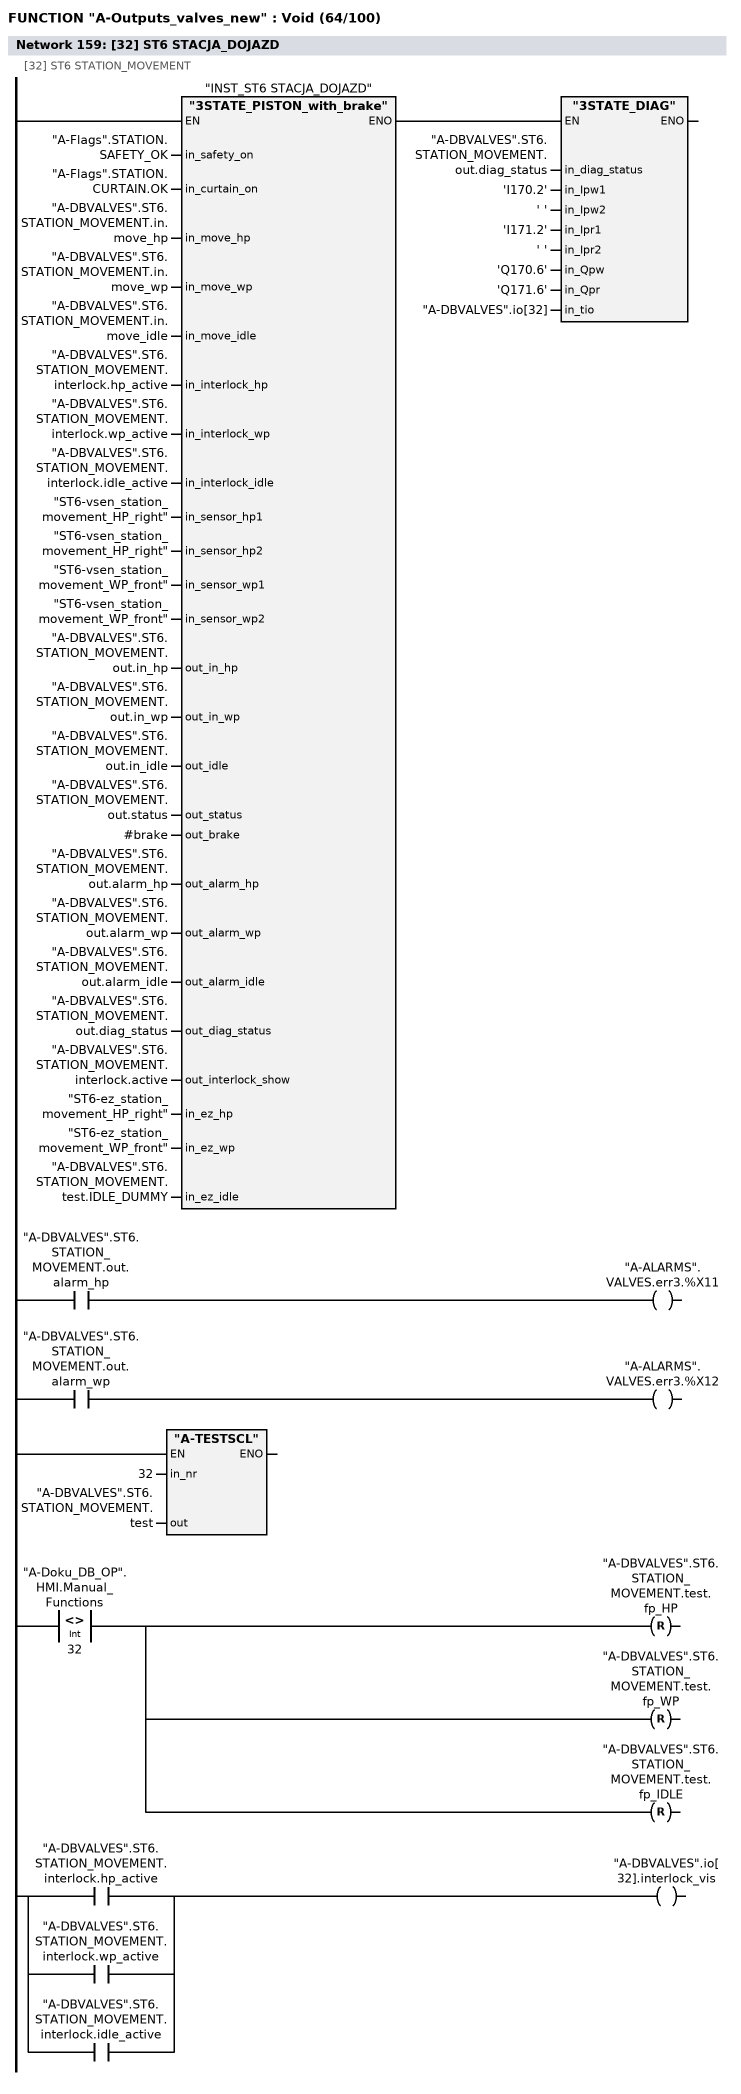
      CALL "3STATE_PISTON_with_brake", "INST_ST6 STACJA_DOJAZD"
      (  in_safety_on                := "A-Flags".STATION.SAFETY_OK ,
         in_curtain_on               := "A-Flags".STATION.CURTAIN.OK ,
         in_move_hp                  := "A-DBVALVES".ST6.STATION_MOVEMENT.in.move_hp ,
         in_move_wp                  := "A-DBVALVES".ST6.STATION_MOVEMENT.in.move_wp ,
         in_move_idle                := "A-DBVALVES".ST6.STATION_MOVEMENT.in.move_idle ,
         in_interlock_hp             := "A-DBVALVES".ST6.STATION_MOVEMENT.interlock.hp_active ,
         in_interlock_wp             := "A-DBVALVES".ST6.STATION_MOVEMENT.interlock.wp_active ,
         in_interlock_idle           := "A-DBVALVES".ST6.STATION_MOVEMENT.interlock.idle_active ,
         in_sensor_hp1               := "ST6-vsen_station_movement_HP_right" ,
         in_sensor_hp2               := "ST6-vsen_station_movement_HP_right" ,
         in_sensor_wp1               := "ST6-vsen_station_movement_WP_front" ,
         in_sensor_wp2               := "ST6-vsen_station_movement_WP_front" ,
         out_in_hp                   := "A-DBVALVES".ST6.STATION_MOVEMENT.out.in_hp ,
         out_in_wp                   := "A-DBVALVES".ST6.STATION_MOVEMENT.out.in_wp ,
         out_idle                    := "A-DBVALVES".ST6.STATION_MOVEMENT.out.in_idle ,
         out_status                  := "A-DBVALVES".ST6.STATION_MOVEMENT.out.status ,
         out_brake                   := #brake ,
         out_alarm_hp                := "A-DBVALVES".ST6.STATION_MOVEMENT.out.alarm_hp ,
         out_alarm_wp                := "A-DBVALVES".ST6.STATION_MOVEMENT.out.alarm_wp ,
         out_alarm_idle              := "A-DBVALVES".ST6.STATION_MOVEMENT.out.alarm_idle ,
         out_diag_status             := "A-DBVALVES".ST6.STATION_MOVEMENT.out.diag_status ,
         out_interlock_show          := "A-DBVALVES".ST6.STATION_MOVEMENT.interlock.active ,
         in_ez_hp                    := "ST6-ez_station_movement_HP_right" ,
         in_ez_wp                    := "ST6-ez_station_movement_WP_front" ,
         in_ez_idle                  := "A-DBVALVES".ST6.STATION_MOVEMENT.test.IDLE_DUMMY
      );

      CALL "3STATE_DIAG"
      (  in_diag_status              := "A-DBVALVES".ST6.STATION_MOVEMENT.out.diag_status ,
         in_Ipw1                     := 'I170.2' ,
         in_Ipw2                     := ' ' ,
         in_Ipr1                     := 'I171.2' ,
         in_Ipr2                     := ' ' ,
         in_Qpw                      := 'Q170.6' ,
         in_Qpr                      := 'Q171.6' ,
         in_tio                      := "A-DBVALVES".io[32]
      );

      A "A-DBVALVES".ST6.STATION_MOVEMENT.out.alarm_hp;
      = "A-ALARMS".VALVES.err3.%X11;

      A "A-DBVALVES".ST6.STATION_MOVEMENT.out.alarm_wp;
      = "A-ALARMS".VALVES.err3.%X12;

      CALL "A-TESTSCL"
      (  in_nr                       := 32 ,
         out                         := "A-DBVALVES".ST6.STATION_MOVEMENT.test
      );

      A(;
      L "A-Doku_DB_OP".HMI.Manual_Functions;
      L 32;
      <>I;
      );
      R "A-DBVALVES".ST6.STATION_MOVEMENT.test.fp_HP;
      R "A-DBVALVES".ST6.STATION_MOVEMENT.test.fp_WP;
      R "A-DBVALVES".ST6.STATION_MOVEMENT.test.fp_IDLE;

      O "A-DBVALVES".ST6.STATION_MOVEMENT.interlock.hp_active;
      O "A-DBVALVES".ST6.STATION_MOVEMENT.interlock.wp_active;
      O "A-DBVALVES".ST6.STATION_MOVEMENT.interlock.idle_active;
      = "A-DBVALVES".io[32].interlock_vis;
NETWORK
TITLE = -

NETWORK
TITLE = [33] ST6 STACJA_MALY_SKOK - HP
//[33] ST6 STATION_SMALL_STEP - HP
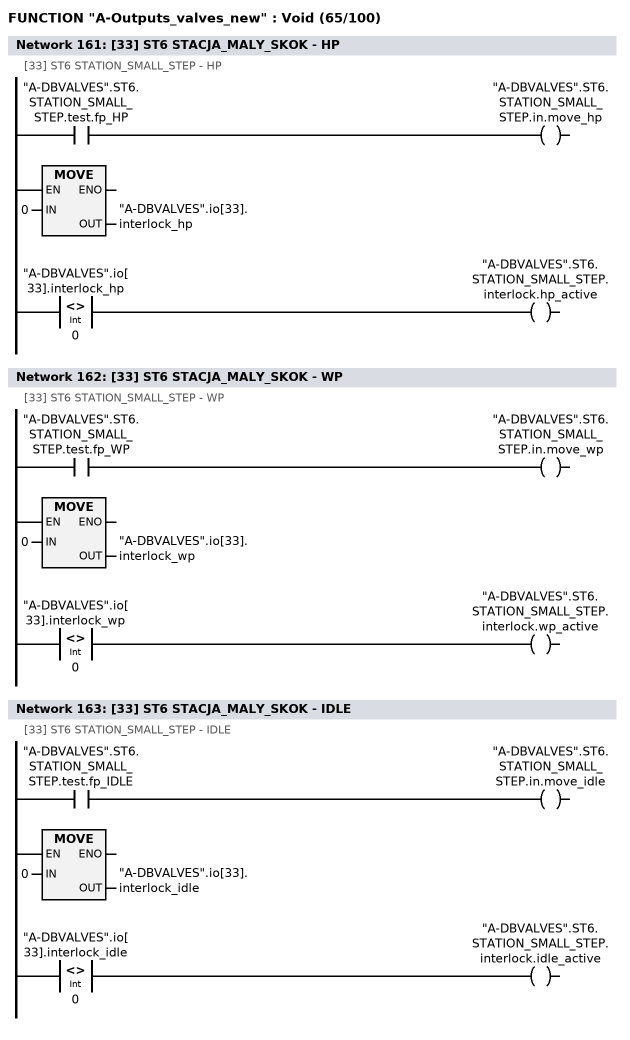
      O "A-DBVALVES".ST6.STATION_SMALL_STEP.test.fp_HP;
//    O     "A-Flags".STATION.IN_HP_STEP
      = "A-DBVALVES".ST6.STATION_SMALL_STEP.in.move_hp;

// Interlock hp
      L 0;
      T "A-DBVALVES".io[33].interlock_hp;

//{INTERLOCK_HP33}

      A(;
      L "A-DBVALVES".io[33].interlock_hp;
      L 0;
      <>I;
      );
      = "A-DBVALVES".ST6.STATION_SMALL_STEP.interlock.hp_active;
NETWORK
TITLE = [33] ST6 STACJA_MALY_SKOK - WP
//[33] ST6 STATION_SMALL_STEP - WP
      O "A-DBVALVES".ST6.STATION_SMALL_STEP.test.fp_WP;
      = "A-DBVALVES".ST6.STATION_SMALL_STEP.in.move_wp;

// Interlock wp
      L 0;
      T "A-DBVALVES".io[33].interlock_wp;

//{INTERLOCK_WP33}

      A(;
      L "A-DBVALVES".io[33].interlock_wp;
      L 0;
      <>I;
      );
      = "A-DBVALVES".ST6.STATION_SMALL_STEP.interlock.wp_active;
NETWORK
TITLE = [33] ST6 STACJA_MALY_SKOK - IDLE
//[33] ST6 STATION_SMALL_STEP - IDLE
      O "A-DBVALVES".ST6.STATION_SMALL_STEP.test.fp_IDLE;
      = "A-DBVALVES".ST6.STATION_SMALL_STEP.in.move_idle;

// Interlock idle
      L 0;
      T "A-DBVALVES".io[33].interlock_idle;

//{INTERLOCK_IDLE33}

      A(;
      L "A-DBVALVES".io[33].interlock_idle;
      L 0;
      <>I;
      );
      = "A-DBVALVES".ST6.STATION_SMALL_STEP.interlock.idle_active;
NETWORK
TITLE = [33] ST6 STACJA_MALY_SKOK
//[33] ST6 STATION_SMALL_STEP
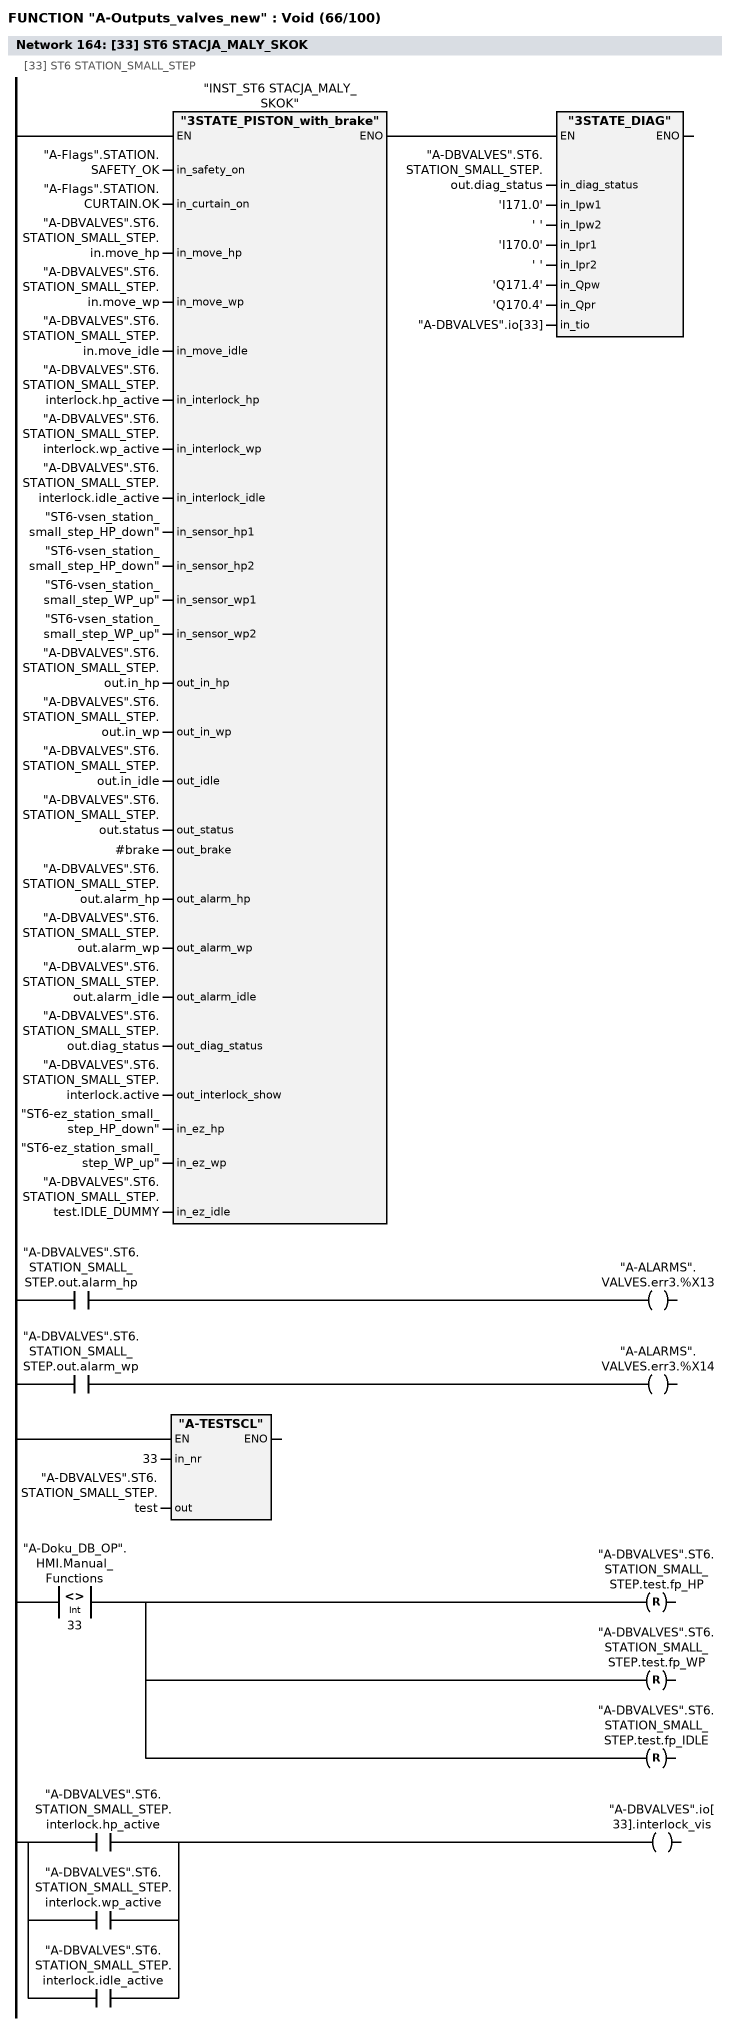
      CALL "3STATE_PISTON_with_brake", "INST_ST6 STACJA_MALY_SKOK"
      (  in_safety_on                := "A-Flags".STATION.SAFETY_OK ,
         in_curtain_on               := "A-Flags".STATION.CURTAIN.OK ,
         in_move_hp                  := "A-DBVALVES".ST6.STATION_SMALL_STEP.in.move_hp ,
         in_move_wp                  := "A-DBVALVES".ST6.STATION_SMALL_STEP.in.move_wp ,
         in_move_idle                := "A-DBVALVES".ST6.STATION_SMALL_STEP.in.move_idle ,
         in_interlock_hp             := "A-DBVALVES".ST6.STATION_SMALL_STEP.interlock.hp_active ,
         in_interlock_wp             := "A-DBVALVES".ST6.STATION_SMALL_STEP.interlock.wp_active ,
         in_interlock_idle           := "A-DBVALVES".ST6.STATION_SMALL_STEP.interlock.idle_active ,
         in_sensor_hp1               := "ST6-vsen_station_small_step_HP_down" ,
         in_sensor_hp2               := "ST6-vsen_station_small_step_HP_down" ,
         in_sensor_wp1               := "ST6-vsen_station_small_step_WP_up" ,
         in_sensor_wp2               := "ST6-vsen_station_small_step_WP_up" ,
         out_in_hp                   := "A-DBVALVES".ST6.STATION_SMALL_STEP.out.in_hp ,
         out_in_wp                   := "A-DBVALVES".ST6.STATION_SMALL_STEP.out.in_wp ,
         out_idle                    := "A-DBVALVES".ST6.STATION_SMALL_STEP.out.in_idle ,
         out_status                  := "A-DBVALVES".ST6.STATION_SMALL_STEP.out.status ,
         out_brake                   := #brake ,
         out_alarm_hp                := "A-DBVALVES".ST6.STATION_SMALL_STEP.out.alarm_hp ,
         out_alarm_wp                := "A-DBVALVES".ST6.STATION_SMALL_STEP.out.alarm_wp ,
         out_alarm_idle              := "A-DBVALVES".ST6.STATION_SMALL_STEP.out.alarm_idle ,
         out_diag_status             := "A-DBVALVES".ST6.STATION_SMALL_STEP.out.diag_status ,
         out_interlock_show          := "A-DBVALVES".ST6.STATION_SMALL_STEP.interlock.active ,
         in_ez_hp                    := "ST6-ez_station_small_step_HP_down" ,
         in_ez_wp                    := "ST6-ez_station_small_step_WP_up" ,
         in_ez_idle                  := "A-DBVALVES".ST6.STATION_SMALL_STEP.test.IDLE_DUMMY
      );

      CALL "3STATE_DIAG"
      (  in_diag_status              := "A-DBVALVES".ST6.STATION_SMALL_STEP.out.diag_status ,
         in_Ipw1                     := 'I171.0' ,
         in_Ipw2                     := ' ' ,
         in_Ipr1                     := 'I170.0' ,
         in_Ipr2                     := ' ' ,
         in_Qpw                      := 'Q171.4' ,
         in_Qpr                      := 'Q170.4' ,
         in_tio                      := "A-DBVALVES".io[33]
      );

      A "A-DBVALVES".ST6.STATION_SMALL_STEP.out.alarm_hp;
      = "A-ALARMS".VALVES.err3.%X13;

      A "A-DBVALVES".ST6.STATION_SMALL_STEP.out.alarm_wp;
      = "A-ALARMS".VALVES.err3.%X14;

      CALL "A-TESTSCL"
      (  in_nr                       := 33 ,
         out                         := "A-DBVALVES".ST6.STATION_SMALL_STEP.test
      );

      A(;
      L "A-Doku_DB_OP".HMI.Manual_Functions;
      L 33;
      <>I;
      );
      R "A-DBVALVES".ST6.STATION_SMALL_STEP.test.fp_HP;
      R "A-DBVALVES".ST6.STATION_SMALL_STEP.test.fp_WP;
      R "A-DBVALVES".ST6.STATION_SMALL_STEP.test.fp_IDLE;

      O "A-DBVALVES".ST6.STATION_SMALL_STEP.interlock.hp_active;
      O "A-DBVALVES".ST6.STATION_SMALL_STEP.interlock.wp_active;
      O "A-DBVALVES".ST6.STATION_SMALL_STEP.interlock.idle_active;
      = "A-DBVALVES".io[33].interlock_vis;
NETWORK
TITLE = -

NETWORK
TITLE = [34] ST6 STACJA_DUZY_SKOK - HP
//[34] ST6 STATION_BIG_STEP - HP
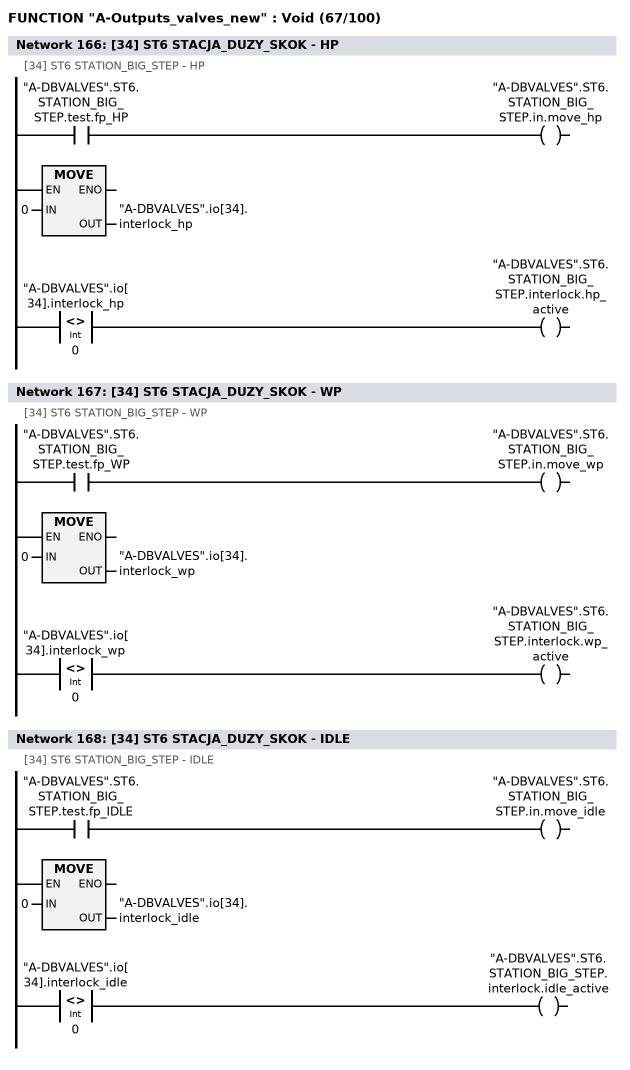
      O "A-DBVALVES".ST6.STATION_BIG_STEP.test.fp_HP;
//    O     "A-Flags".STATION.IN_HP_STEP
      = "A-DBVALVES".ST6.STATION_BIG_STEP.in.move_hp;

// Interlock hp
      L 0;
      T "A-DBVALVES".io[34].interlock_hp;

//{INTERLOCK_HP34}

      A(;
      L "A-DBVALVES".io[34].interlock_hp;
      L 0;
      <>I;
      );
      = "A-DBVALVES".ST6.STATION_BIG_STEP.interlock.hp_active;
NETWORK
TITLE = [34] ST6 STACJA_DUZY_SKOK - WP
//[34] ST6 STATION_BIG_STEP - WP
      O "A-DBVALVES".ST6.STATION_BIG_STEP.test.fp_WP;
      = "A-DBVALVES".ST6.STATION_BIG_STEP.in.move_wp;

// Interlock wp
      L 0;
      T "A-DBVALVES".io[34].interlock_wp;

//{INTERLOCK_WP34}

      A(;
      L "A-DBVALVES".io[34].interlock_wp;
      L 0;
      <>I;
      );
      = "A-DBVALVES".ST6.STATION_BIG_STEP.interlock.wp_active;
NETWORK
TITLE = [34] ST6 STACJA_DUZY_SKOK - IDLE
//[34] ST6 STATION_BIG_STEP - IDLE
      O "A-DBVALVES".ST6.STATION_BIG_STEP.test.fp_IDLE;
      = "A-DBVALVES".ST6.STATION_BIG_STEP.in.move_idle;

// Interlock idle
      L 0;
      T "A-DBVALVES".io[34].interlock_idle;

//{INTERLOCK_IDLE34}

      A(;
      L "A-DBVALVES".io[34].interlock_idle;
      L 0;
      <>I;
      );
      = "A-DBVALVES".ST6.STATION_BIG_STEP.interlock.idle_active;
NETWORK
TITLE = [34] ST6 STACJA_DUZY_SKOK
//[34] ST6 STATION_BIG_STEP
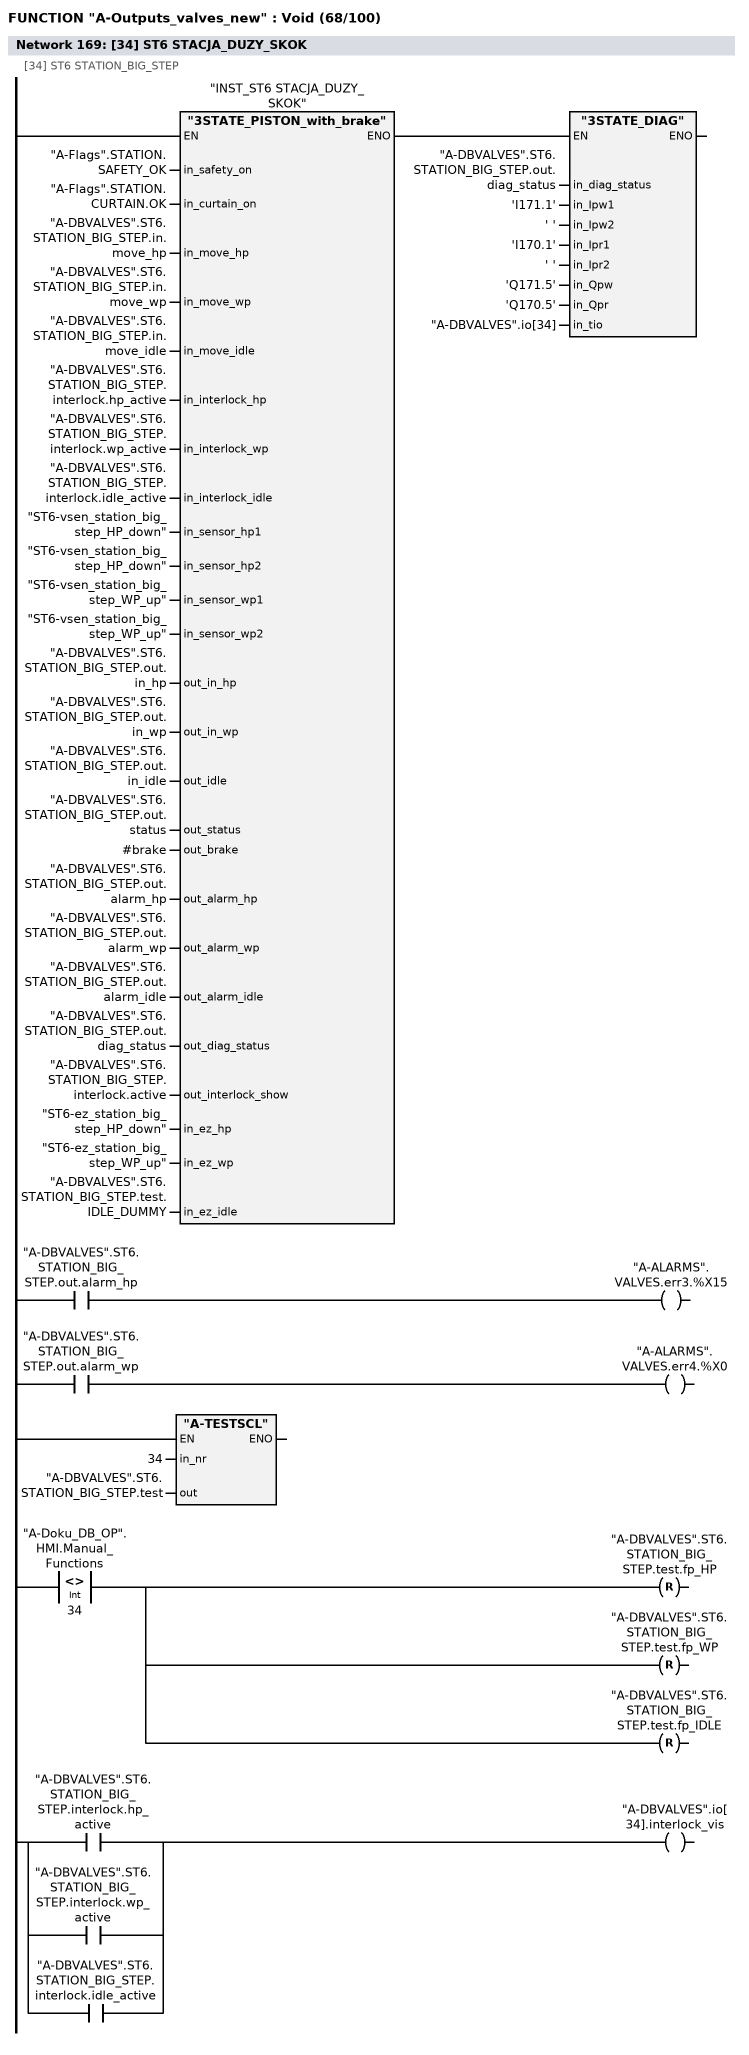
      CALL "3STATE_PISTON_with_brake", "INST_ST6 STACJA_DUZY_SKOK"
      (  in_safety_on                := "A-Flags".STATION.SAFETY_OK ,
         in_curtain_on               := "A-Flags".STATION.CURTAIN.OK ,
         in_move_hp                  := "A-DBVALVES".ST6.STATION_BIG_STEP.in.move_hp ,
         in_move_wp                  := "A-DBVALVES".ST6.STATION_BIG_STEP.in.move_wp ,
         in_move_idle                := "A-DBVALVES".ST6.STATION_BIG_STEP.in.move_idle ,
         in_interlock_hp             := "A-DBVALVES".ST6.STATION_BIG_STEP.interlock.hp_active ,
         in_interlock_wp             := "A-DBVALVES".ST6.STATION_BIG_STEP.interlock.wp_active ,
         in_interlock_idle           := "A-DBVALVES".ST6.STATION_BIG_STEP.interlock.idle_active ,
         in_sensor_hp1               := "ST6-vsen_station_big_step_HP_down" ,
         in_sensor_hp2               := "ST6-vsen_station_big_step_HP_down" ,
         in_sensor_wp1               := "ST6-vsen_station_big_step_WP_up" ,
         in_sensor_wp2               := "ST6-vsen_station_big_step_WP_up" ,
         out_in_hp                   := "A-DBVALVES".ST6.STATION_BIG_STEP.out.in_hp ,
         out_in_wp                   := "A-DBVALVES".ST6.STATION_BIG_STEP.out.in_wp ,
         out_idle                    := "A-DBVALVES".ST6.STATION_BIG_STEP.out.in_idle ,
         out_status                  := "A-DBVALVES".ST6.STATION_BIG_STEP.out.status ,
         out_brake                   := #brake ,
         out_alarm_hp                := "A-DBVALVES".ST6.STATION_BIG_STEP.out.alarm_hp ,
         out_alarm_wp                := "A-DBVALVES".ST6.STATION_BIG_STEP.out.alarm_wp ,
         out_alarm_idle              := "A-DBVALVES".ST6.STATION_BIG_STEP.out.alarm_idle ,
         out_diag_status             := "A-DBVALVES".ST6.STATION_BIG_STEP.out.diag_status ,
         out_interlock_show          := "A-DBVALVES".ST6.STATION_BIG_STEP.interlock.active ,
         in_ez_hp                    := "ST6-ez_station_big_step_HP_down" ,
         in_ez_wp                    := "ST6-ez_station_big_step_WP_up" ,
         in_ez_idle                  := "A-DBVALVES".ST6.STATION_BIG_STEP.test.IDLE_DUMMY
      );

      CALL "3STATE_DIAG"
      (  in_diag_status              := "A-DBVALVES".ST6.STATION_BIG_STEP.out.diag_status ,
         in_Ipw1                     := 'I171.1' ,
         in_Ipw2                     := ' ' ,
         in_Ipr1                     := 'I170.1' ,
         in_Ipr2                     := ' ' ,
         in_Qpw                      := 'Q171.5' ,
         in_Qpr                      := 'Q170.5' ,
         in_tio                      := "A-DBVALVES".io[34]
      );

      A "A-DBVALVES".ST6.STATION_BIG_STEP.out.alarm_hp;
      = "A-ALARMS".VALVES.err3.%X15;

      A "A-DBVALVES".ST6.STATION_BIG_STEP.out.alarm_wp;
      = "A-ALARMS".VALVES.err4.%X0;

      CALL "A-TESTSCL"
      (  in_nr                       := 34 ,
         out                         := "A-DBVALVES".ST6.STATION_BIG_STEP.test
      );

      A(;
      L "A-Doku_DB_OP".HMI.Manual_Functions;
      L 34;
      <>I;
      );
      R "A-DBVALVES".ST6.STATION_BIG_STEP.test.fp_HP;
      R "A-DBVALVES".ST6.STATION_BIG_STEP.test.fp_WP;
      R "A-DBVALVES".ST6.STATION_BIG_STEP.test.fp_IDLE;

      O "A-DBVALVES".ST6.STATION_BIG_STEP.interlock.hp_active;
      O "A-DBVALVES".ST6.STATION_BIG_STEP.interlock.wp_active;
      O "A-DBVALVES".ST6.STATION_BIG_STEP.interlock.idle_active;
      = "A-DBVALVES".io[34].interlock_vis;
NETWORK
TITLE = -

NETWORK
TITLE = [35] ST6 PIN - HP
//[35] ST6 PIN - HP
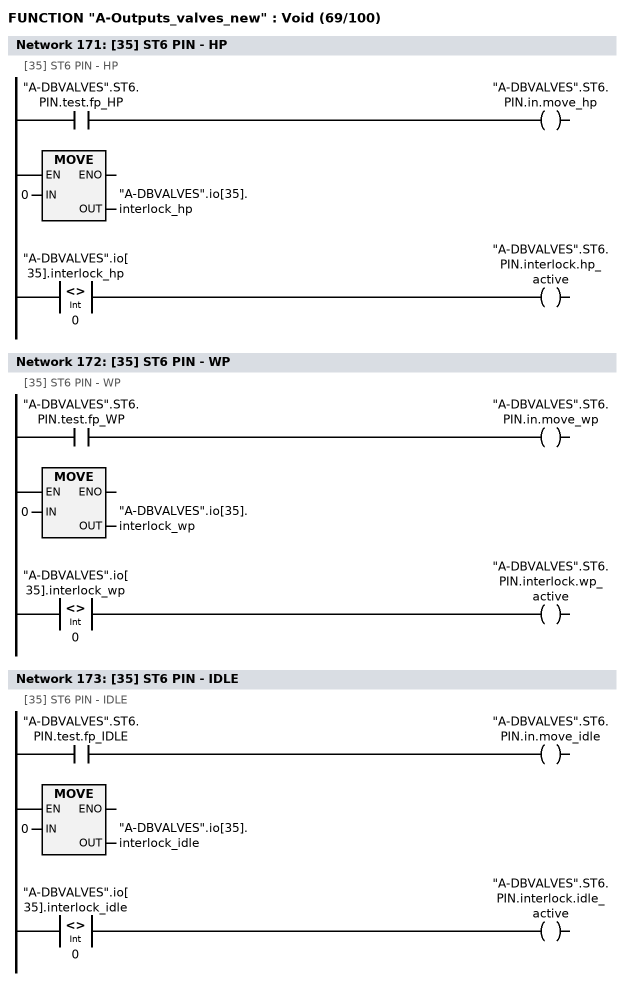
      O "A-DBVALVES".ST6.PIN.test.fp_HP;
//    O     "A-Flags".STATION.IN_HP_STEP
      = "A-DBVALVES".ST6.PIN.in.move_hp;

// Interlock hp
      L 0;
      T "A-DBVALVES".io[35].interlock_hp;

//{INTERLOCK_HP35}

      A(;
      L "A-DBVALVES".io[35].interlock_hp;
      L 0;
      <>I;
      );
      = "A-DBVALVES".ST6.PIN.interlock.hp_active;
NETWORK
TITLE = [35] ST6 PIN - WP
//[35] ST6 PIN - WP
      O "A-DBVALVES".ST6.PIN.test.fp_WP;
      = "A-DBVALVES".ST6.PIN.in.move_wp;

// Interlock wp
      L 0;
      T "A-DBVALVES".io[35].interlock_wp;

//{INTERLOCK_WP35}

      A(;
      L "A-DBVALVES".io[35].interlock_wp;
      L 0;
      <>I;
      );
      = "A-DBVALVES".ST6.PIN.interlock.wp_active;
NETWORK
TITLE = [35] ST6 PIN - IDLE
//[35] ST6 PIN - IDLE
      O "A-DBVALVES".ST6.PIN.test.fp_IDLE;
      = "A-DBVALVES".ST6.PIN.in.move_idle;

// Interlock idle
      L 0;
      T "A-DBVALVES".io[35].interlock_idle;

//{INTERLOCK_IDLE35}

      A(;
      L "A-DBVALVES".io[35].interlock_idle;
      L 0;
      <>I;
      );
      = "A-DBVALVES".ST6.PIN.interlock.idle_active;
NETWORK
TITLE = [35] ST6 PIN
//[35] ST6 PIN
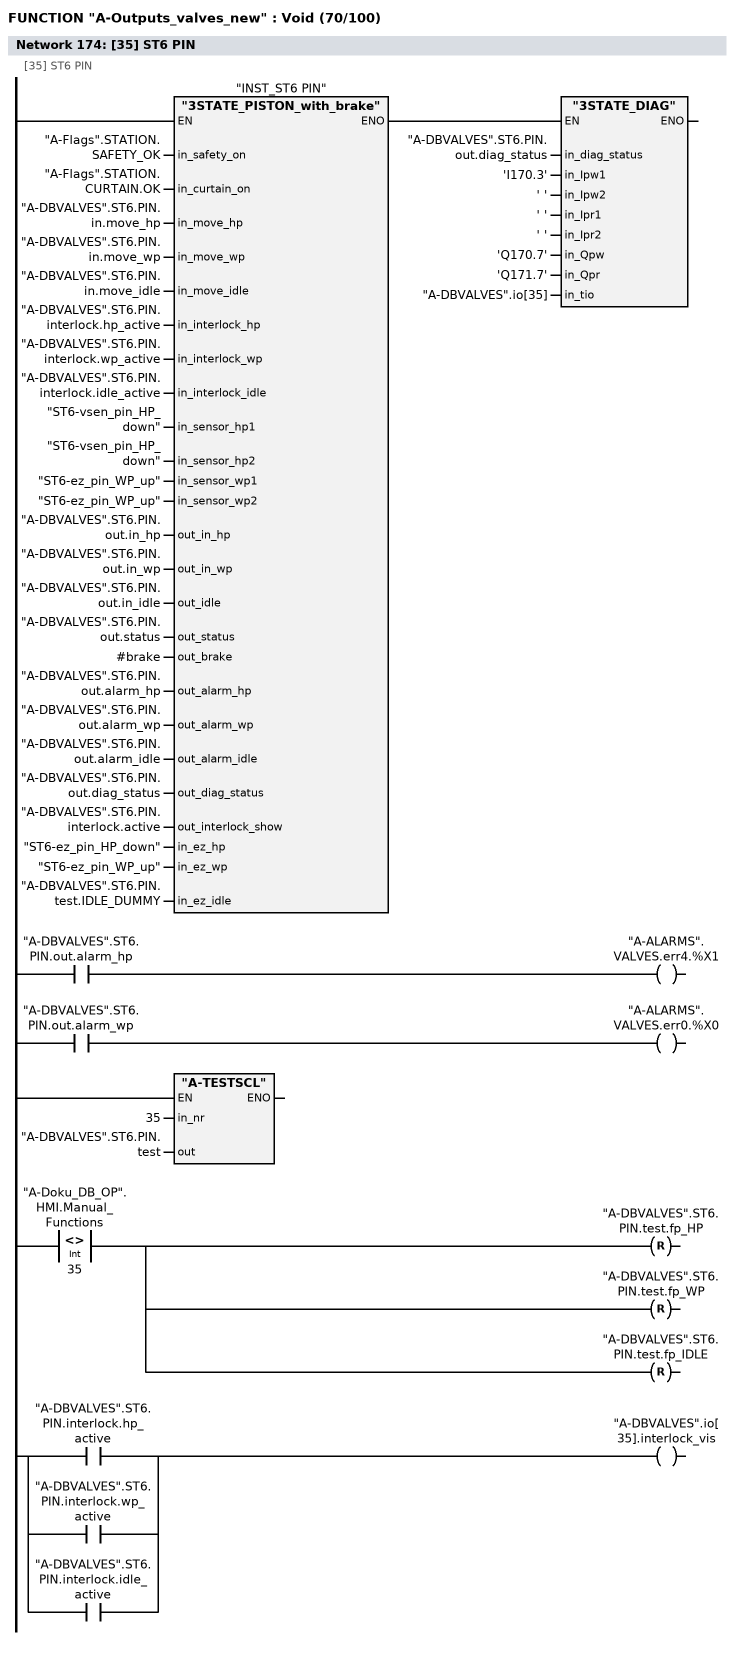
      CALL "3STATE_PISTON_with_brake", "INST_ST6 PIN"
      (  in_safety_on                := "A-Flags".STATION.SAFETY_OK ,
         in_curtain_on               := "A-Flags".STATION.CURTAIN.OK ,
         in_move_hp                  := "A-DBVALVES".ST6.PIN.in.move_hp ,
         in_move_wp                  := "A-DBVALVES".ST6.PIN.in.move_wp ,
         in_move_idle                := "A-DBVALVES".ST6.PIN.in.move_idle ,
         in_interlock_hp             := "A-DBVALVES".ST6.PIN.interlock.hp_active ,
         in_interlock_wp             := "A-DBVALVES".ST6.PIN.interlock.wp_active ,
         in_interlock_idle           := "A-DBVALVES".ST6.PIN.interlock.idle_active ,
         in_sensor_hp1               := "ST6-vsen_pin_HP_down" ,
         in_sensor_hp2               := "ST6-vsen_pin_HP_down" ,
         in_sensor_wp1               := "ST6-ez_pin_WP_up" ,
         in_sensor_wp2               := "ST6-ez_pin_WP_up" ,
         out_in_hp                   := "A-DBVALVES".ST6.PIN.out.in_hp ,
         out_in_wp                   := "A-DBVALVES".ST6.PIN.out.in_wp ,
         out_idle                    := "A-DBVALVES".ST6.PIN.out.in_idle ,
         out_status                  := "A-DBVALVES".ST6.PIN.out.status ,
         out_brake                   := #brake ,
         out_alarm_hp                := "A-DBVALVES".ST6.PIN.out.alarm_hp ,
         out_alarm_wp                := "A-DBVALVES".ST6.PIN.out.alarm_wp ,
         out_alarm_idle              := "A-DBVALVES".ST6.PIN.out.alarm_idle ,
         out_diag_status             := "A-DBVALVES".ST6.PIN.out.diag_status ,
         out_interlock_show          := "A-DBVALVES".ST6.PIN.interlock.active ,
         in_ez_hp                    := "ST6-ez_pin_HP_down" ,
         in_ez_wp                    := "ST6-ez_pin_WP_up" ,
         in_ez_idle                  := "A-DBVALVES".ST6.PIN.test.IDLE_DUMMY
      );

      CALL "3STATE_DIAG"
      (  in_diag_status              := "A-DBVALVES".ST6.PIN.out.diag_status ,
         in_Ipw1                     := 'I170.3' ,
         in_Ipw2                     := ' ' ,
         in_Ipr1                     := ' ' ,
         in_Ipr2                     := ' ' ,
         in_Qpw                      := 'Q170.7' ,
         in_Qpr                      := 'Q171.7' ,
         in_tio                      := "A-DBVALVES".io[35]
      );

      A "A-DBVALVES".ST6.PIN.out.alarm_hp;
      = "A-ALARMS".VALVES.err4.%X1;

      A "A-DBVALVES".ST6.PIN.out.alarm_wp;
      = "A-ALARMS".VALVES.err0.%X0;

      CALL "A-TESTSCL"
      (  in_nr                       := 35 ,
         out                         := "A-DBVALVES".ST6.PIN.test
      );

      A(;
      L "A-Doku_DB_OP".HMI.Manual_Functions;
      L 35;
      <>I;
      );
      R "A-DBVALVES".ST6.PIN.test.fp_HP;
      R "A-DBVALVES".ST6.PIN.test.fp_WP;
      R "A-DBVALVES".ST6.PIN.test.fp_IDLE;

      O "A-DBVALVES".ST6.PIN.interlock.hp_active;
      O "A-DBVALVES".ST6.PIN.interlock.wp_active;
      O "A-DBVALVES".ST6.PIN.interlock.idle_active;
      = "A-DBVALVES".io[35].interlock_vis;
NETWORK
TITLE = -

NETWORK
TITLE = [36] ST7L MIECZ_SKOSNY_DOJAZD - HP
//[36] ST7L SWORD_ANGLE_MOVEMENT - HP
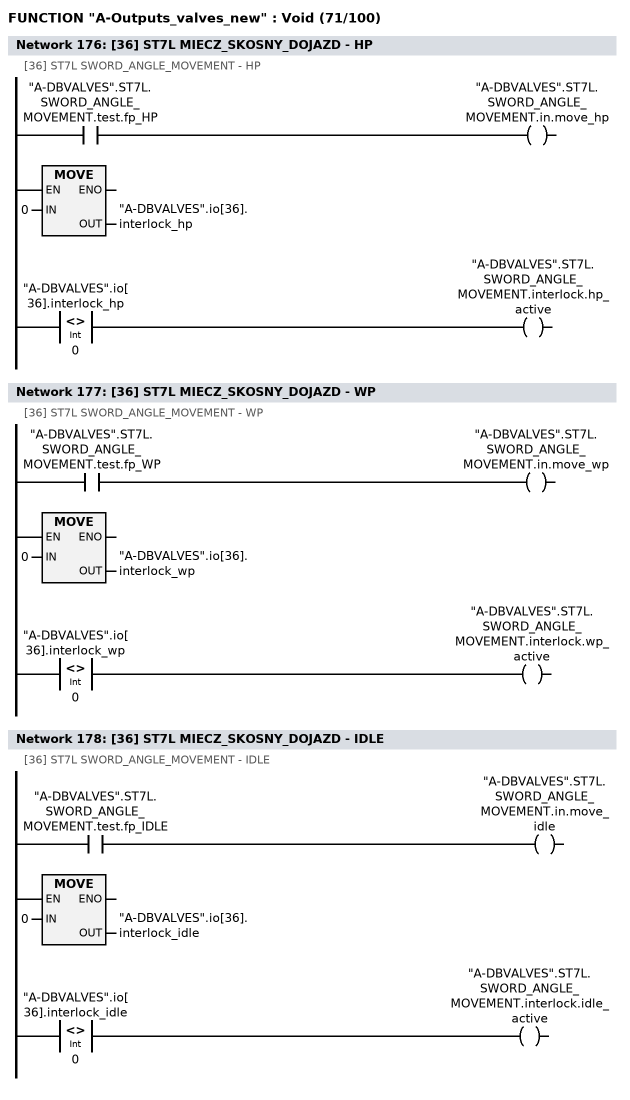
      O "A-DBVALVES".ST7L.SWORD_ANGLE_MOVEMENT.test.fp_HP;
//    O     "A-Flags".STATION.IN_HP_STEP
      = "A-DBVALVES".ST7L.SWORD_ANGLE_MOVEMENT.in.move_hp;

// Interlock hp
      L 0;
      T "A-DBVALVES".io[36].interlock_hp;

//{INTERLOCK_HP36}

      A(;
      L "A-DBVALVES".io[36].interlock_hp;
      L 0;
      <>I;
      );
      = "A-DBVALVES".ST7L.SWORD_ANGLE_MOVEMENT.interlock.hp_active;
NETWORK
TITLE = [36] ST7L MIECZ_SKOSNY_DOJAZD - WP
//[36] ST7L SWORD_ANGLE_MOVEMENT - WP
      O "A-DBVALVES".ST7L.SWORD_ANGLE_MOVEMENT.test.fp_WP;
      = "A-DBVALVES".ST7L.SWORD_ANGLE_MOVEMENT.in.move_wp;

// Interlock wp
      L 0;
      T "A-DBVALVES".io[36].interlock_wp;

//{INTERLOCK_WP36}

      A(;
      L "A-DBVALVES".io[36].interlock_wp;
      L 0;
      <>I;
      );
      = "A-DBVALVES".ST7L.SWORD_ANGLE_MOVEMENT.interlock.wp_active;
NETWORK
TITLE = [36] ST7L MIECZ_SKOSNY_DOJAZD - IDLE
//[36] ST7L SWORD_ANGLE_MOVEMENT - IDLE
      O "A-DBVALVES".ST7L.SWORD_ANGLE_MOVEMENT.test.fp_IDLE;
      = "A-DBVALVES".ST7L.SWORD_ANGLE_MOVEMENT.in.move_idle;

// Interlock idle
      L 0;
      T "A-DBVALVES".io[36].interlock_idle;

//{INTERLOCK_IDLE36}

      A(;
      L "A-DBVALVES".io[36].interlock_idle;
      L 0;
      <>I;
      );
      = "A-DBVALVES".ST7L.SWORD_ANGLE_MOVEMENT.interlock.idle_active;
NETWORK
TITLE = [36] ST7L MIECZ_SKOSNY_DOJAZD
//[36] ST7L SWORD_ANGLE_MOVEMENT
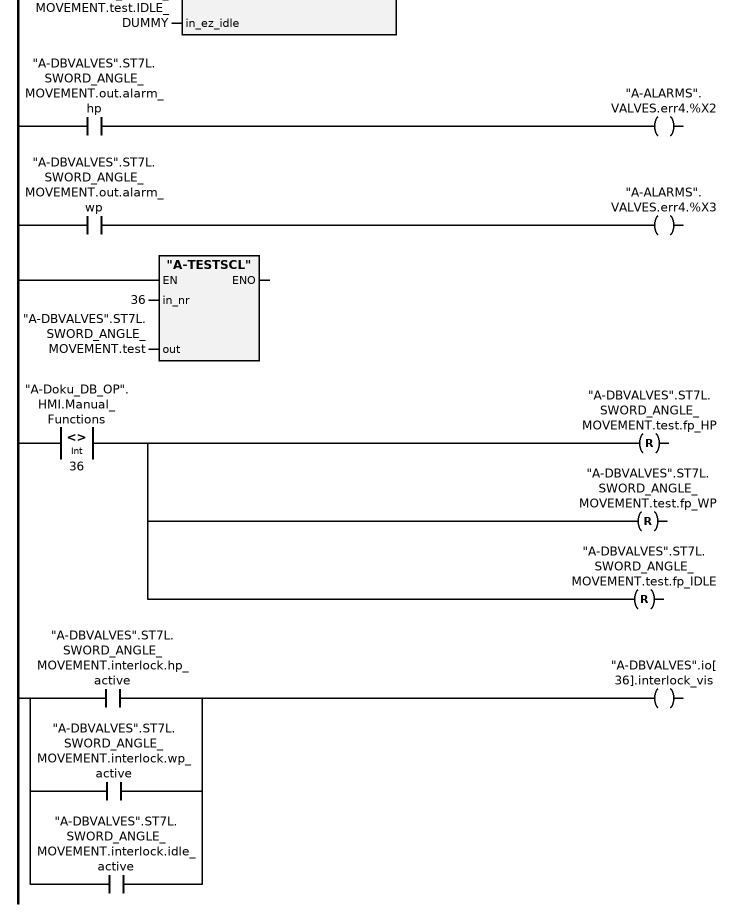
      CALL "3STATE_PISTON_with_brake", "INST_ST7L MIECZ_SKOSNY_DOJAZD"
      (  in_safety_on                := "A-Flags".STATION.SAFETY_OK ,
         in_curtain_on               := "A-Flags".STATION.CURTAIN.OK ,
         in_move_hp                  := "A-DBVALVES".ST7L.SWORD_ANGLE_MOVEMENT.in.move_hp ,
         in_move_wp                  := "A-DBVALVES".ST7L.SWORD_ANGLE_MOVEMENT.in.move_wp ,
         in_move_idle                := "A-DBVALVES".ST7L.SWORD_ANGLE_MOVEMENT.in.move_idle ,
         in_interlock_hp             := "A-DBVALVES".ST7L.SWORD_ANGLE_MOVEMENT.interlock.hp_active ,
         in_interlock_wp             := "A-DBVALVES".ST7L.SWORD_ANGLE_MOVEMENT.interlock.wp_active ,
         in_interlock_idle           := "A-DBVALVES".ST7L.SWORD_ANGLE_MOVEMENT.interlock.idle_active ,
         in_sensor_hp1               := "ST7L-vsen_sword_angle_movement_HP_right" ,
         in_sensor_hp2               := "ST7L-vsen_sword_angle_movement_HP_right" ,
         in_sensor_wp1               := "ST7L-vsen_sword_angle_movement_WP_front" ,
         in_sensor_wp2               := "ST7L-vsen_sword_angle_movement_WP_front" ,
         out_in_hp                   := "A-DBVALVES".ST7L.SWORD_ANGLE_MOVEMENT.out.in_hp ,
         out_in_wp                   := "A-DBVALVES".ST7L.SWORD_ANGLE_MOVEMENT.out.in_wp ,
         out_idle                    := "A-DBVALVES".ST7L.SWORD_ANGLE_MOVEMENT.out.in_idle ,
         out_status                  := "A-DBVALVES".ST7L.SWORD_ANGLE_MOVEMENT.out.status ,
         out_brake                   := #brake ,
         out_alarm_hp                := "A-DBVALVES".ST7L.SWORD_ANGLE_MOVEMENT.out.alarm_hp ,
         out_alarm_wp                := "A-DBVALVES".ST7L.SWORD_ANGLE_MOVEMENT.out.alarm_wp ,
         out_alarm_idle              := "A-DBVALVES".ST7L.SWORD_ANGLE_MOVEMENT.out.alarm_idle ,
         out_diag_status             := "A-DBVALVES".ST7L.SWORD_ANGLE_MOVEMENT.out.diag_status ,
         out_interlock_show          := "A-DBVALVES".ST7L.SWORD_ANGLE_MOVEMENT.interlock.active ,
         in_ez_hp                    := "ST7L-ez_sword_angle_movement_HP_right" ,
         in_ez_wp                    := "ST7L-ez_sword_angle_movement_WP_front" ,
         in_ez_idle                  := "A-DBVALVES".ST7L.SWORD_ANGLE_MOVEMENT.test.IDLE_DUMMY
      );

      CALL "3STATE_DIAG"
      (  in_diag_status              := "A-DBVALVES".ST7L.SWORD_ANGLE_MOVEMENT.out.diag_status ,
         in_Ipw1                     := 'I140.0' ,
         in_Ipw2                     := ' ' ,
         in_Ipr1                     := 'I141.0' ,
         in_Ipr2                     := ' ' ,
         in_Qpw                      := 'Q140.5' ,
         in_Qpr                      := 'Q141.5' ,
         in_tio                      := "A-DBVALVES".io[36]
      );

      A "A-DBVALVES".ST7L.SWORD_ANGLE_MOVEMENT.out.alarm_hp;
      = "A-ALARMS".VALVES.err4.%X2;

      A "A-DBVALVES".ST7L.SWORD_ANGLE_MOVEMENT.out.alarm_wp;
      = "A-ALARMS".VALVES.err4.%X3;

      CALL "A-TESTSCL"
      (  in_nr                       := 36 ,
         out                         := "A-DBVALVES".ST7L.SWORD_ANGLE_MOVEMENT.test
      );

      A(;
      L "A-Doku_DB_OP".HMI.Manual_Functions;
      L 36;
      <>I;
      );
      R "A-DBVALVES".ST7L.SWORD_ANGLE_MOVEMENT.test.fp_HP;
      R "A-DBVALVES".ST7L.SWORD_ANGLE_MOVEMENT.test.fp_WP;
      R "A-DBVALVES".ST7L.SWORD_ANGLE_MOVEMENT.test.fp_IDLE;

      O "A-DBVALVES".ST7L.SWORD_ANGLE_MOVEMENT.interlock.hp_active;
      O "A-DBVALVES".ST7L.SWORD_ANGLE_MOVEMENT.interlock.wp_active;
      O "A-DBVALVES".ST7L.SWORD_ANGLE_MOVEMENT.interlock.idle_active;
      = "A-DBVALVES".io[36].interlock_vis;
NETWORK
TITLE = -

NETWORK
TITLE = [37] ST7L MIECZ_PROSTY_DOJAZD - HP
//[37] ST7L SWORD_STRAIGHT_MOVEMENT - HP
